// TwinCAT 3 PLC project IDPLC
// ProgramVersion: 3.1.4024.12
// libraries:
//   Tc2_Drive, * (Beckhoff Automation GmbH)
//   Tc2_EtherCAT, * (Beckhoff Automation GmbH)
//   Tc2_Math, * (Beckhoff Automation GmbH)
//   Tc2_MC2, * (Beckhoff Automation GmbH)
//   Tc2_NC, * (Beckhoff Automation GmbH)
//   Tc2_NcDrive, * (Beckhoff Automation GmbH)
//   Tc2_SerialCom, * (Beckhoff Automation GmbH)
//   Tc2_Standard, * (Beckhoff Automation GmbH)
//   Tc2_System, * (Beckhoff Automation GmbH)
//   Tc2_Utilities, * (Beckhoff Automation GmbH)
//   Tc3_Module, * (Beckhoff Automation GmbH)
// project tree:
//   DUTs/ DUT.TcDUT, DUT_SENSOR_DATAS_1.TcDUT, DUT_SENSOR_DATAS_8.TcDUT, DUT_SENSOR_DATAS_2.TcDUT, DUT_SENSOR_DATAS_3.TcDUT, DUT_SENSOR_DATAS_4.TcDUT, DUT_SENSOR_DATAS_5.TcDUT, DUT_SENSOR_DATAS_6.TcDUT, DUT_SENSOR_DATAS_7.TcDUT, Struct_M_Compensation.TcDUT, Struct_M_lakeshore.TcDUT
//   GVLs/ Global_Variables.TcGVL, Variable_Configuration.TcGVL
//   / PlcTask.TcTTO, RecipeManager.TcRMO (not stored)
//   POUs/0.UserMode/ F_GetSysTime.TcPOU, UserMode.TcPOU
//   POUs/1.CarrierMode/GapMode/ BCGapMode.TcPOU, GapMode.TcPOU
//   POUs/1.CarrierMode/SingleCarrierMode/ SingleCarrierMode.TcPOU
//   POUs/2.SingleMotorMode/DebugMode/ DebugMode.TcPOU
//   POUs/2.SingleMotorMode/TaperMode/ TaperMode.TcPOU
//   POUs/CommonFB/ExternFB/ FB_LedShow.TcPOU, FB_PlcEmergencyStop.TcPOU
//   POUs/CommonFB/MainFB/ FB_CoupleAxis.TcPOU, FB_DecoupleAxis.TcPOU, FB_Move.TcPOU, FB_Power.TcPOU, FB_SetAxisPosition.TcPOU, FB_Stop.TcPOU
//   POUs/ MAIN.TcPOU
//   POUs/MainPRG/ FB_CheckCoupleStatus.TcPOU
//   POUs/RS232/ BackgroundEL.TcPOU, FB_SerialCom.TcPOU

CONFIGURATION IDPLC
    RESOURCE PLC ON TwinCAT3
        TASK PlcTask(INTERVAL := T#10ms, PRIORITY := 20);
        PROGRAM MAIN WITH PlcTask : MAIN;
    END_RESOURCE
END_CONFIGURATION

// ---- DUTs/DUT.TcDUT
TYPE DUT :
STRUCT
	Encoder:LREAL;
	LeftTop:LREAL;
END_STRUCT
END_TYPE

// ---- DUTs/DUT_SENSOR_DATAS_1.TcDUT
TYPE DUT_SENSOR_DATAS_1 :
UNION
	data_lreal:REAL;
	data_byte:ARRAY[0..3] OF BYTE;
END_UNION
END_TYPE

// ---- DUTs/DUT_SENSOR_DATAS_8.TcDUT
TYPE DUT_SENSOR_DATAS_8 :
UNION
	data_lreal:REAL;
	data_byte:ARRAY[0..3] OF BYTE;
END_UNION
END_TYPE

// ---- DUTs/DUT_SENSOR_DATAS_2.TcDUT
TYPE DUT_SENSOR_DATAS_2 :
UNION
	data_lreal:REAL;
	data_byte:ARRAY[0..3] OF BYTE;
END_UNION
END_TYPE

// ---- DUTs/DUT_SENSOR_DATAS_3.TcDUT
TYPE DUT_SENSOR_DATAS_3 :
UNION
	data_lreal:REAL;
	data_byte:ARRAY[0..3] OF BYTE;
END_UNION
END_TYPE

// ---- DUTs/DUT_SENSOR_DATAS_4.TcDUT
TYPE DUT_SENSOR_DATAS_4 :
UNION
	data_lreal:REAL;
	data_byte:ARRAY[0..3] OF BYTE;
END_UNION
END_TYPE

// ---- DUTs/DUT_SENSOR_DATAS_5.TcDUT
TYPE DUT_SENSOR_DATAS_5 :
UNION
	data_lreal:REAL;
	data_byte:ARRAY[0..3] OF BYTE;
END_UNION
END_TYPE

// ---- DUTs/DUT_SENSOR_DATAS_6.TcDUT
TYPE DUT_SENSOR_DATAS_6 :
UNION
	data_lreal:REAL;
	data_byte:ARRAY[0..3] OF BYTE;
END_UNION
END_TYPE

// ---- DUTs/DUT_SENSOR_DATAS_7.TcDUT
TYPE DUT_SENSOR_DATAS_7 :
UNION
	data_lreal:REAL;
	data_byte:ARRAY[0..3] OF BYTE;
END_UNION
END_TYPE

// ---- DUTs/Struct_M_Compensation.TcDUT
TYPE Struct_M_Compensation :
STRUCT
	Encoder:LREAL;
	LeftTop:LREAL;
	RightTop:LREAL;
	LeftBottom:LREAL;
	RightBottom:LREAL;
	InRange:BOOL;
END_STRUCT
END_TYPE

// ---- DUTs/Struct_M_lakeshore.TcDUT
TYPE Struct_M_lakeshore :
STRUCT
	Temperature:LREAL;(*Celsius*)
	Resistance:LREAL;
END_STRUCT
END_TYPE

// ---- GVLs/Global_Variables.TcGVL
//{attribute 'Tc2GvlVarNames'}
VAR_GLOBAL
(*IDControl Ready*)
	IDControlReady:BOOL;
(*Error Massage*)
	Error:BOOL;
	ErrorID:DINT;
	ErrorDescription:STRING;
(*加载配方参数*)
	LoadRecipeParameters:BOOL;
	loadParametersDone:BOOL;
(*设置光栅bias done *)	
	PositionBiasDone:BOOL;
(*回程差*)
	HysteresisError:LREAL;
(*Drive Status*)
	DriveStatus:DINT;//1:Drive Ready;2:Axis is in operation;0:Others
(*光栅漂移误差阈值*)
	LEDriftErrorThreshold:LREAL:=0.001;
(*Lag Distance threshold*)
	PosDiff_LeftTopLin: LREAL:=0.5;
	PosDiff_RightTopLin:LREAL:=0.5;
	PosDiff_LeftBottomLin:LREAL:=0.5;
	PosDiff_RightBottomLin:LREAL:=0.5;
(*UserMode Threshold*)
	Threshold_UserTopPos: LREAL:=0.5;
	Threshold_UserBottomPos: LREAL:=0.5;
	Threshold_UserLeftPos: LREAL:=0.5;
	Threshold_UserRightPos: LREAL:=0.5;
	Threshold_UserTopVelo: LREAL:=0.5;
	Threshold_UserBottomVelo: LREAL:=0.5;
	Threshold_UserLeftVelo: LREAL:=0.5;
	Threshold_UserRightVelo: LREAL:=0.5;
	//
	Range_UserTaperPos:LREAL:=4.01;
	Range_UserTaperVelo:LREAL:=1.01;
	//Diff_TaperLeftPos:LREAL:=0.01;
	//Diff_TaperLeftVelo:LREAL:=0.2;
	//Diff_TaperRightPos:LREAL:=0.05;
	//Diff_TaperRightVelo:LREAL:=0.5;
	//Taper_BeyondRangePositive:BOOL;
	//Diff_TaperTopPos:LREAL:=0.05;
	//Diff_TaperBottomPos:LREAL:=0.05;
	//Taper_BeyondRangeNegtive:BOOL;
(*BCGap Threshold*)
	Threshold_BCTopPos: LREAL:=0.5;
	Threshold_BCBottomPos: LREAL:=0.5;
	Threshold_BCLeftPos: LREAL:=0.5;
	Threshold_BCRightPos: LREAL:=0.5;
	Threshold_BCTopVelo: LREAL:=0.5;
	Threshold_BCBottomVelo: LREAL:=0.5;
	Threshold_BCLeftVelo: LREAL:=0.5;
	Threshold_BCRightVelo: LREAL:=0.5;
(*DebugMode Threshold*)
	Threshold_TopPos_Debug: LREAL:=4;
	Threshold_BottomPos_Debug: LREAL:=4;
	Threshold_LeftPos_Debug: LREAL:=4;
	Threshold_RightPos_Debug: LREAL:=4;
(*Taper Mode Threshold*)
	Range_TaperPos:LREAL:=5.01;
	Range_TaperVelo:LREAL:=1.01;
	Threshold_TaperLeftPos:LREAL:=0.01;
	Threshold_TaperLeftVelo:LREAL:=0.2;
	Threshold_TaperRightPos:LREAL:=0.05;
	Threshold_TaperRightVelo:LREAL:=0.5;
	Taper_BeyondRangePositive:BOOL;
	Threshold_TaperTopPos:LREAL:=0.05;
	Threshold_TaperBottomPos:LREAL:=0.05;
	Taper_BeyondRangeNegtive:BOOL;
(*SingleCarrierMode threshold*)
	Threshold_TopPos_SingleCarrier: LREAL:=2;
	Threshold_BottomPos_SingleCarrier: LREAL:=2;
	Threshold_LeftPos_SingleCarrier: LREAL:=2;
	Threshold_RightPos_SingleCarrier: LREAL:=2;
	Threshold_TopVelo_SingleCarrier: LREAL:=2;
	Threshold_BottomVelo_SingleCarrier: LREAL:=2;
	Threshold_LeftVelo_SingleCarrier: LREAL:=2;
	Threshold_RightVelo_SingleCarrier: LREAL:=2;
(*Compensation Value*)
	M_Compensation:ARRAY[1..18] OF Struct_M_Compensation
:=[
(Encoder:=0,	LeftTop:=0,	RightTop:=0,		LeftBottom:=0,	RightBottom:=0,	InRange:=FALSE),
(Encoder:=5.5,	LeftTop:=5.5,	RightTop:=5.5,	LeftBottom:=5.5,	RightBottom:=5.5,	InRange:=FALSE),
(Encoder:=6.0,	LeftTop:=6.0,	RightTop:=6.0,	LeftBottom:=6.0,	RightBottom:=6.0,	InRange:=FALSE),
(Encoder:=6.5,	LeftTop:=6.5,	RightTop:=6.5,	LeftBottom:=6.5,	RightBottom:=6.5,	InRange:=FALSE),
(Encoder:=7.5,	LeftTop:=7.5,	RightTop:=7.5,	LeftBottom:=7.5,	RightBottom:=7.5,	InRange:=FALSE),
(Encoder:=8.5,	LeftTop:=8.5,	RightTop:=8.5,	LeftBottom:=8.5,	RightBottom:=8.5,	InRange:=FALSE),
(Encoder:=9.5,	LeftTop:=9.5,	RightTop:=9.5,	LeftBottom:=9.5,	RightBottom:=9.5,	InRange:=FALSE),
(Encoder:=10.5,	LeftTop:=10.5,	RightTop:=10.5,	LeftBottom:=10.5,	RightBottom:=10.5,		InRange:=FALSE),
(Encoder:=11.5,	LeftTop:=11.5,	RightTop:=11.5,	LeftBottom:=11.5,	RightBottom:=11.5,		InRange:=FALSE),
(Encoder:=30.0,	LeftTop:=30.0,	RightTop:=30.0,	LeftBottom:=30.0,	RightBottom:=30.0,		InRange:=FALSE),
(Encoder:=100.0,	LeftTop:=100.0,	RightTop:=100.0,	LeftBottom:=100.0,	RightBottom:=100.0,		InRange:=FALSE),
(Encoder:=110.0,	LeftTop:=110.0,	RightTop:=110.0,	LeftBottom:=110.0,	RightBottom:=110.0,		InRange:=FALSE),
(Encoder:=120.0,	LeftTop:=120.0,	RightTop:=120.0,	LeftBottom:=120.0,	RightBottom:=120.0,		InRange:=FALSE),
(Encoder:=130.0,	LeftTop:=130.0,	RightTop:=130.0,	LeftBottom:=130.0,	RightBottom:=130.0,		InRange:=FALSE),
(Encoder:=140.0,	LeftTop:=140.0,	RightTop:=140.0,	LeftBottom:=140.0,	RightBottom:=140.0,		InRange:=FALSE),
(Encoder:=150.0,	LeftTop:=150.0,	RightTop:=150.0,	LeftBottom:=150.0,	RightBottom:=150.0,		InRange:=FALSE),
(Encoder:=160.0,	LeftTop:=160.0,	RightTop:=160.0,	LeftBottom:=160.0,	RightBottom:=160.0,		InRange:=FALSE),
(Encoder:=3000.001,	LeftTop:=3000.001,	RightTop:=3000.001,		LeftBottom:=3000.001,	RightBottom:=3000.001,	InRange:=FALSE)];

(*simulation OR NOT*)
	simulation:BOOL;
(*USELinearEncoeder*)
	USELinearEncoder:BOOL:=TRUE;
(*restartTwinCAT*)
	m_restartTC:BOOL;
(*Plc_EmergencyStop *)
	Plc_EmergencyStop  AT %Q*:BOOL:=TRUE;
(*硬急停*)
	Hardware_EmergencyStop :BOOL:=TRUE;
(*LED*)
	Led_Run  AT %Q*:BOOL;
	Led_Error  AT %Q*:BOOL;
(*LimitSwitch*)
	LS_LeftTop_Top  :BOOL;
	LS_LeftTop_Bottom  :BOOL;
	LS_RightTop_Top  :BOOL;
	LS_RightTop_Bottom  :BOOL;
	LS_LeftBottom_Top  :BOOL;
	LS_LeftBottom_Bottom  :BOOL;
	LS_RightBottom_Top :BOOL;
	LS_RightBottom_Bottom  :BOOL;
	Unreach_LS_Top:BOOL;
	Unreach_LS_Bottom:BOOL;
(*kill switch*)
	KS_LeftTop_Far_Contact1:BOOL;
	KS_LeftTop_Far_Contact2:BOOL;
	KS_RightTop_Far_Contact1:BOOL;
	KS_RightTop_Far_Contact2:BOOL;
	KS_LeftBottom_Far_Contact1:BOOL;
	KS_LeftBottom_Far_Contact2:BOOL;
	KS_RightBottom_Far_Contact1:BOOL;
	KS_RightBottom_Far_Contact2:BOOL;
	
	KS_LeftTop_Near_Contact1:BOOL;
	KS_LeftTop_Near_Contact2:BOOL;
	KS_RightTop_Near_Contact1:BOOL;
	KS_RightTop_Near_Contact2:BOOL;
	KS_LeftBottom_Near_Contact1:BOOL;
	KS_LeftBottom_Near_Contact2:BOOL;
	KS_RightBottom_Near_Contact1:BOOL;
	KS_RightBottom_Near_Contact2:BOOL;
(*E-STOP*)
	KS_CabinetEmergency_contact1:BOOL;
	KS_CabinetEmergency_contact2:BOOL;
	KS_handEmergency1_Contact1:BOOL;
	KS_handEmergency1_Contact2:BOOL;
	KS_handEmergency2_Contact1:BOOL;
	KS_handEmergency2_Contact2:BOOL;
	KS_softEmergency2_Contact:BOOL;
(*aixs_ref*)
	LeftTopLin: axis_ref;
	RightTopLin:axis_ref;
	LeftBottomLin:axis_ref;
	RightBottomLin:axis_ref;
(*axis Position*)
	Pos_LeftTopLin: LREAL;
	Pos_RightTopLin:LREAL;
	Pos_LeftBottomLin:LREAL;
	Pos_RightBottomLin:LREAL;
(*********)
	LB_TestRecord:LREAL;
	RB_TestRecord:LREAL;
(*axis Velocity*)
	Velo_LeftTopLin: LREAL;
	Velo_RightTopLin:LREAL;
	Velo_LeftBottomLin:LREAL;
	Velo_RightBottomLin:LREAL;
(*Lag Distance*)
	PosDiff_LeftTopLin_actual: LREAL;
	PosDiff_RightTopLin_actual:LREAL;
	PosDiff_LeftBottomLin_actual:LREAL;
	PosDiff_RightBottomLin_actual:LREAL;
(********************Gap Mode*************************)
(**)
	GapPositionActual:LREAL;
	GapVelocityActual:LREAL;
	GapMoveIndicator:DINT:=0;
	(*1=OPEN;0=NOTMOVE;-1=CLOSE*)
(******************Taper Mode**************************)
(*Taper*)
	TaperPositionActual:LREAL;
	TaperVelocityActual:LREAL;
	TaperMoveIndicator:DINT:=0;
	(*1=OPEN;0=NOTMOVE;-1=CLOSE*)
(*****************singleCarrier Mode*******************************)
(**)
	TopPositionActual:LREAL;
	TopVelocityActual:LREAL;
	BottomPositionActual:LREAL;
	BottomVelocityActual:LREAL;
	TopMoveIndicator:DINT:=0;
	(*1=OPEN;0=NOTMOVE;-1=CLOSE*)
	BottomMoveIndicator:DINT:=0;
	(*1=OPEN;0=NOTMOVE;-1=CLOSE*)
(******************DebugMode & BCGapMode*****************************)
	LeftTopLinMoveIndicator:DINT:=0;
	(*1=OPEN;0=NOTMOVE;-1=CLOSE*)
	LeftBottomLinMoveIndicator:DINT:=0;
	(*1=OPEN;0=NOTMOVE;-1=CLOSE*)
	RightTopLinMoveIndicator:DINT:=0;
	(*1=OPEN;0=NOTMOVE;-1=CLOSE*)
	RightBottomLinMoveIndicator:DINT:=0;
	(*1=OPEN;0=NOTMOVE;-1=CLOSE*)
(******************Gap&SingleCarrier***********************************)
	Diff_TopPos_actual: LREAL;
	Diff_BottomPos_actual: LREAL;
	Diff_LeftPos_actual: LREAL;
	Diff_RightPos_actual: LREAL;
	Diff_TopVelo_actual:  LREAL;
	Diff_BottomVelo_actual: LREAL;
	Diff_LeftVelo_actual: LREAL;
	Diff_RightVelo_actual:  LREAL;

(******************BCGap Mode***********************************)
	Diff_BCTopPos_actual: LREAL;
	Diff_BCBottomPos_actual: LREAL;
	Diff_BCLeftPos_actual: LREAL;
	Diff_BCRightPos_actual: LREAL;
	Diff_BCTopVelo_actual:  LREAL;
	Diff_BCBottomVelo_actual: LREAL;
	Diff_BCLeftVelo_actual: LREAL;
	Diff_BCRightVelo_actual:  LREAL;
(******************UserMode*********************)
	Diff_UserTopPos_actual: LREAL;
	Diff_UserBottomPos_actual: LREAL;
	Diff_UserLeftPos_actual: LREAL;
	Diff_UserRightPos_actual: LREAL;
	Diff_UserTopVelo_actual:  LREAL;
	Diff_UserBottomVelo_actual: LREAL;
	Diff_UserLeftVelo_actual: LREAL;
	Diff_UserRightVelo_actual:  LREAL;
	TaperOrNot:BOOL;
	UserTaperPositionActual:LREAL;
	UserTaperVelocityActual:LREAL;
(***********************Power status and couple statatus***********************)
	st_Power:BOOL;
	st_Couple:DINT;
(************************FB***********************)
	FB_Power:FB_Power;
	FB_PlcEmergencyStop: FB_PlcEmergencyStop;
	FB_CheckCoupleStatus:FB_CheckCoupleStatus;
	FB_Move:FB_Move;
	FB_Stop:FB_Stop;
	FB_DecoupleAxis:FB_DecoupleAxis;
	FB_CoupleAxis: FB_CoupleAxis;
(********************²¹³¥GapÄ£Ê½£¬µ¥Öá²¹³¥Êý¾Ý************************)
	(*ÊÇ·ñ²¹³¥*)
	USE_SingleAxis_Compensation:BOOL:=TRUE;
	Mdut:ARRAY[1..2] OF DUT:=
	[(Encoder:=2.0,	LeftTop:=2.3000),
	(Encoder:=2.0,	LeftTop:=2.3000)];


	M_CompensationNumber:INT;
	M_DisplayNumber:INT;
	(*Conpensation Position Target*)
	LeftTopLinPositionNew:LREAL;
	LeftBottomLinPositionNew:LREAL;
	RightTopLinPositionNew:LREAL;
	RightBottomLinPositionNew:LREAL;
	(*考虑到回程差后，运动到临时位置*)
	LeftTopLinPositionNew_temporary :LREAL;
	LeftBottomLinPositionNew_temporary:LREAL;
	RightTopLinPositionNew_temporary:LREAL;
	RightBottomLinPositionNew_temporary:LREAL;
	(*Display Position*)
	LeftTopLinPositionDisplay:LREAL;
	LeftBottomLinPositionDisplay:LREAL;
	RightTopLinPositionDisplay:LREAL;
	RightBottomLinPositionDisplay:LREAL;
	(*Display Velocity*)
	LeftTopLinVelocityDisplay:LREAL;
	LeftBottomLinVelocityDisplay:LREAL;
	RightTopLinVelocityDisplay:LREAL;
	RightBottomLinVelocityDisplay:LREAL;
	(*temperature sensors*)
	thermocouple AT %I*:ARRAY[1..12]OF  DINT;
	shieldPt100  AT %I*:ARRAY[1..12]OF INT;
	thermocouple_Celsius:ARRAY[1..12]OF  LREAL;
	shieldPt100_Celsius  :ARRAY[1..12]OF LREAL;
	huoer_Celsius AT %I* :ARRAY[1..3]OF INT;
	(**)
	lakeshorePt100  AT %I*:ARRAY[1..12]OF INT;(*16*×èÖµ*)
	lakeshorePt100_Resistance :ARRAY[1..12]OF LREAL;(*ÉãÊÏÎÂ¶È*)
	lakeshorePt100_Celsius  :ARRAY[1..12]OF LREAL;(*ÉãÊÏÎÂ¶È*)
	temperatureCompensationValue:LREAL:=6;
	testSensors  AT %I*:ARRAY[1..4]OF INT;

(*Test No.184*)
	Struct_M_lakeshore_168:ARRAY[1..52] OF Struct_M_lakeshore:=[(Temperature:=-255.02072961,	Resistance:=19394.22709513),
														       (Temperature:=-254.05045152,	Resistance:=17654.92429047),
														       (Temperature:=-253.07744087,	Resistance:=16151.62683151),
														       (Temperature:=-252.00959324,	Resistance:=14730.57326945),
														       (Temperature:=-250.42495220,	Resistance:=12968.55015283),
														       (Temperature:=-248.82081761,	Resistance:=11509.89960915),
														       (Temperature:=-247.21174565,	Resistance:=10296.55197911),
														       (Temperature:=-245.58891366,	Resistance:=9270.75571767),
														       (Temperature:=-243.96558907,	Resistance:=8400.62569432),
														       (Temperature:=-242.14354329,	Resistance:=7573.26483503),
														       (Temperature:=-240.02689351,	Resistance:=6767.17126789),
														       (Temperature:=-237.01618411,	Resistance:=5838.58514549),
														       (Temperature:=-234.00593745,	Resistance:=5101.58555065),
														       (Temperature:=-230.99752410,	Resistance:=4505.18214539),
														       (Temperature:=-228.00173193,	Resistance:=4017.09732257),
														       (Temperature:=-224.99947745,	Resistance:=3609.02040601),
														       (Temperature:=-223.00692641,	Resistance:=3374.28026471),
														       (Temperature:=-218.01660226,	Resistance:=2884.61719537),
														       (Temperature:=-213.02574325,	Resistance:=2501.58514940),
														       (Temperature:=-208.03560884,	Resistance:=2195.64012040),
														       (Temperature:=-203.04420176,	Resistance:=1946.81103230),
														       (Temperature:=-198.05275449,	Resistance:=1741.06206884),
														       (Temperature:=-193.06103279,	Resistance:=1568.92560629),
														       (Temperature:=-188.06248282,	Resistance:=1422.92395120),
														       (Temperature:=-183.06714354,	Resistance:=1298.17958491),
														       (Temperature:=-178.06870827,	Resistance:=1190.47468069),
														       (Temperature:=-173.07068956,	Resistance:=1096.60468916),
														       (Temperature:=-163.08053594,	Resistance:=942.07281950),
														       (Temperature:=-153.08718985,	Resistance:=820.42837839),
														       (Temperature:=-143.08487641,	Resistance:=722.56760466),
														       (Temperature:=-133.08398781,	Resistance:=642.67848926),
														       (Temperature:=-123.08745222,	Resistance:=576.45895597),
														       (Temperature:=-113.09120089,	Resistance:=520.90762376),
														       (Temperature:=-103.09942915,	Resistance:=473.74837218),
														       (Temperature:=-93.10598968,		Resistance:=433.38294834),
														       (Temperature:=-83.10392915,		Resistance:=398.41968464),
														       (Temperature:=-73.10228709,		Resistance:=368.09301028),
														       (Temperature:=-63.10299621,		Resistance:=341.43424414),
														       (Temperature:=-53.11519681,		Resistance:=318.02847824),
														       (Temperature:=-43.10742807	,	Resistance:=297.22485607),
														       (Temperature:=-33.10726812,		Resistance:=278.69871028),
														       (Temperature:=-23.11858134,		Resistance:=262.15834948),
														       (Temperature:=-13.10195090,		Resistance:=247.23616978),
														       (Temperature:=-3.11184252,		Resistance:=233.79708047),
														       (Temperature:=6.89903472,		Resistance:=221.61300733),
														       (Temperature:=16.89346621,		Resistance:=210.54967929),
														       (Temperature:=26.90358952,		Resistance:=200.45587628),
														       (Temperature:=36.88287604,		Resistance:=191.25204791),
														       (Temperature:=41.88872196,		Resistance:=186.92616816),
														       (Temperature:=46.88480694,		Resistance:=182.78432099),
														       (Temperature:=52.87776550,		Resistance:=178.06184409),
														       (Temperature:=56.87370113,		Resistance:=175.01081354)];

(*
Struct_M_lakeshore_168:ARRAY[1..52] OF Struct_M_lakeshore:=(Temperature:=-255.02148584,	Resistance:=17467.51361429),
														       (Temperature:=-254.05229765,	Resistance:=15920.82205731),
														       (Temperature:=-253.07582822,	Resistance:=14578.50586503),
														       (Temperature:=-252.01029408,	Resistance:=13314.83293750),
														       (Temperature:=-250.42593953,	Resistance:=11741.46150061),
														       (Temperature:=-248.82114671,	Resistance:=10435.92048251),
														       (Temperature:=-247.21093179,	Resistance:=9348.73725539),
														       (Temperature:=-245.58869114,	Resistance:=8428.36508630),
														       (Temperature:=-243.96317077,	Resistance:=7645.95382882),
														       (Temperature:=-242.14282659,	Resistance:=6901.52980185),
														       (Temperature:=-240.02565306,	Resistance:=6174.70288700),
														       (Temperature:=-237.01772619,	Resistance:=5337.15935418),
														       (Temperature:=-234.00641032,	Resistance:=4669.94432605),
														       (Temperature:=-230.99638631,	Resistance:=4129.44762482),
														       (Temperature:=-228.00091359,	Resistance:=3686.25091590),
														       (Temperature:=-225.00020456,	Resistance:=3315.69773718),
														       (Temperature:=-223.00791577,	Resistance:=3102.03825436),
														       (Temperature:=-218.01784455,	Resistance:=2655.95765650),
														       (Temperature:=-213.02820409,	Resistance:=2306.30469335),
														       (Temperature:=-208.03707086,	Resistance:=2026.68631979),
														       (Temperature:=-203.04413996,	Resistance:=1798.75031171),
														       (Temperature:=-198.05551086,	Resistance:=1610.35975891),
														       (Temperature:=-193.06273927,	Resistance:=1452.39526661),
														       (Temperature:=-188.05883288,	Resistance:=1318.25592597),
														       (Temperature:=-183.06258538,	Resistance:=1203.56234118),
														       (Temperature:=-178.06718279,	Resistance:=1104.51148216),
														       (Temperature:=-173.07249199,	Resistance:=1018.20332165),
														       (Temperature:=-163.08375191,	Resistance:=875.68114167),
														       (Temperature:=-153.08708895,	Resistance:=763.40014611),
														       (Temperature:=-143.08456026,	Resistance:=673.01413079),
														       (Temperature:=-133.08511977,	Resistance:=599.14558137),
														       (Temperature:=-123.08749266,	Resistance:=537.87435730),
														       (Temperature:=-113.09351200,	Resistance:=486.39730699),
														       (Temperature:=-103.10083499,	Resistance:=442.70701049),
														       (Temperature:=-93.10681179,		Resistance:=405.24490154),
														       (Temperature:=-83.10668364,		Resistance:=372.85251196),
														       (Temperature:=-73.10424427,		Resistance:=344.62377216),
														       (Temperature:=-63.10525050,		Resistance:=319.91272482),
														       (Temperature:=-53.11631884,		Resistance:=298.14326645),
														       (Temperature:=-43.10919062	,	Resistance:=278.79776489),
														       (Temperature:=-33.10718139,		Resistance:=261.57224548),
														       (Temperature:=-23.12143823,		Resistance:=246.17864217),
														       (Temperature:=-13.10564070,		Resistance:=232.27707124),
														       (Temperature:=-3.11271856,		Resistance:=219.77787693),
														       (Temperature:=6.89876028,		Resistance:=208.41568062),
														       (Temperature:=16.88935188,		Resistance:=198.10158580),
														       (Temperature:=26.89992337,		Resistance:=188.70405160),
														       (Temperature:=36.88110394,		Resistance:=180.10572832),
														       (Temperature:=41.88616228,		Resistance:=176.08361784),
														       (Temperature:=46.88372409,		Resistance:=172.21346348),
														       (Temperature:=52.87452959,		Resistance:=167.80352164),
														       (Temperature:=56.87233822,		Resistance:=164.96790544);
*)

(******RS232************)
	RxBufferEL			: ComBuffer;	(* Receive data buffer; used with all receive function blocks *)
	TxBufferEL			: ComBuffer;	(* Transmit data buffer; used with all receive function blocks *)

END_VAR

// ---- GVLs/Variable_Configuration.TcGVL
{attribute 'Tc2GvlVarNames'}
VAR_CONFIG
END_VAR

// ---- POUs/MAIN.TcPOU
PROGRAM MAIN
VAR
	pbGapMode: BOOL:=FALSE;
	pbTaperMode: BOOL:=FALSE;
	pbSingleCarrierMode: BOOL:=FALSE;
	pbDebugMode:BOOL:=FALSE;
	pbBCGapMode:BOOL:=FALSE;
	fb_led_Show: FB_LedShow;
	btn_reset: BOOL;
	CPMU_PLC_Reset: PLC_Reset;
	d_state: DINT;
	CPMU_PLC_Start: PLC_Start;
	powerStatus:BOOL;

(*TwinSAFE*)
	Safe_run AT%Q*:BOOL;
	Err_Ack AT %Q*:BOOL;
	Estop_RunAndRestart AT %Q*:BOOL;
	AX5805_Error_Ack AT %Q*:BOOL;
	Led_Run  AT %Q*:BOOL;
	Led_Error  AT %Q*:BOOL;

	FB_ERROR AT%I*:BOOL;
	COM_ERROR AT%I*:BOOL;
	//OUT_ERROR AT%I*:BOOL;
	Estop_Out AT%I*:BOOL;

	SafeStatus:INT;
	SafePLCRunOK: BOOL;
	fb_ton: TON;
	fb_ton2: TON;
	fb_ton3: TON;
	fb_ton1: TON;
	fb_ton0: TON;
(*IO*)
	el1808_D1  AT%I* :ARRAY[1..8] OF BOOL;
	el1008 AT%I*:BOOL;
	EStopTrig:BOOL;
(*setAxisPosition*)
	SetAxisPosState: INT;
	FB_Set_AxisPosition:FB_SetAxisPosition;
	fb_ton4: TON;
	fb_ton5: TON;
	fb_ton6: TON;
	SerAxisPositionDone: BOOL;

	i: INT;
	j: INT;

(****RS232***)
	fbEL6001	: FB_SerialCom;
	moveDoneLeftTop: BOOL;
	moveDoneRightTop: BOOL;
	moveDoneLeftBottom: BOOL;
	moveDoneRightBottom: BOOL;
	moveDoneAllAxis: BOOL;
	moveStatusLeftTop: BOOL;
	moveStatusRightTop: BOOL;
	moveStatusLeftBottom: BOOL;
	moveStatusRightBottom: BOOL;
	moveStatusAllAxis: BOOL;

(*Torque*)
	Torque_LT AT%I*:INT;
	Torque_RT AT%I*:INT;
	Torque_LB AT%I*:INT;
	Torque_RB AT%I*:INT;
(**)
	btn_setAxisPosition: BOOL;
	ValueSet_LeftTop:LREAL;
	ValueSet_RightTop:LREAL;
	ValueSet_LeftBottom:LREAL;
	ValueSet_RightBottom:LREAL;
(**)
	RestartTC: TC_Restart;
	
(*recipe*)
	RecipeINT:INT;
	RecipeBOOL:BOOL;
	RecipeManCommands: RecipeManCommands;
	SaveParameter : BOOL;  //保存文件
	LoadParameter : BOOL;  //读取文件
	Save_R_TRIG   : R_TRIG;
	Read_R_TRIG   : R_TRIG;
	loadparameterStatus: INT;
	RecipeBOOL2:BOOL;
	ReturnDwordLoad: DWORD;
	InsertionDeviceName:STRING;
(*UserMode*)
	pbUserMode: BOOL:=TRUE;
	EL1904 AT%I* :ARRAY[1..24] OF BOOL;
	setAxisPositionEnable: BOOL;
	state_loadParameters: INT;
	state_setLEPosBias: INT;
	//
	PositionBiasSet:BOOL;
	MC_SetLEPosBias_LeftTop:MC_WriteParameter;
	MC_SetLEPosBias_RightTop:MC_WriteParameter;
	MC_SetLEPosBias_LeftBottom:MC_WriteParameter;
	MC_SetLEPosBias_RightBottom:MC_WriteParameter;
	PositionBias_LeftTop: LREAL:=10.1;
	PositionBias_RightTop: LREAL:=10.2;
	PositionBias_LeftBottom: LREAL:=10.3;
	PositionBias_RightBottom: LREAL:=10.4;

	LoadLEPB_R_TRIG: R_TRIG;
	PositionBiasTON: TON;
	
	//
	OPC_TEST_Bi:BOOL:=TRUE; (*~ (OPC:1:available for OPC Clients) *)
	OPC_TEST_Bi2:BOOL;(*~ (OPC:1:available for OPC Clients) *)
	//
	HasTemperatureSensorOrNot:BOOL;//Only IVU or CPMU
	(*Sensor Reading*)
	Sensor_Reading_1 AT %I*:ARRAY[0..3] OF BYTE;
	Sensor_Reading_2 AT %I*:ARRAY[0..3] OF BYTE;
	Sensor_Reading_3 AT %I*:ARRAY[0..3] OF BYTE;
	Sensor_Reading_4 AT %I*:ARRAY[0..3] OF BYTE;
	Sensor_Reading_5 AT %I*:ARRAY[0..3] OF BYTE;
	Sensor_Reading_6 AT %I*:ARRAY[0..3] OF BYTE;
	Sensor_Reading_7 AT %I*:ARRAY[0..3] OF BYTE;
	Sensor_Reading_8 AT %I*:ARRAY[0..3] OF BYTE;
	Sensor_Reading_DpState AT %I*:USINT;
	Sensor_Reading_ExtDiagFlag AT %I*:BOOL;
	TemperatureSensors_1:LREAL;
	TemperatureSensors_2:LREAL;
	TemperatureSensors_3:LREAL;
	TemperatureSensors_4:LREAL;
	TemperatureSensors_5:LREAL;
	TemperatureSensors_6:LREAL;
	TemperatureSensors_7:LREAL;
	TemperatureSensors_8:LREAL;
	dut_sensor_datas_1:DUT_SENSOR_DATAS_1;
	dut_sensor_datas_2:DUT_SENSOR_DATAS_2;
	dut_sensor_datas_3:DUT_SENSOR_DATAS_3;
	dut_sensor_datas_4:DUT_SENSOR_DATAS_4;
	dut_sensor_datas_5:DUT_SENSOR_DATAS_5;
	dut_sensor_datas_6:DUT_SENSOR_DATAS_6;
	dut_sensor_datas_7:DUT_SENSOR_DATAS_7;
	dut_sensor_datas_8:DUT_SENSOR_DATAS_8;
	//
	temperature_gradient_2_To_1:LREAL;
	temperature_gradient_3_To_2:LREAL;
	temperature_gradient_5_To_4:LREAL;
	temperature_gradient_6_To_5:LREAL;
	temperature_gradient_max:LREAL;
	//
	temperature_average:LREAL;
	A_SetLinearEncoderPositionBias_Enable: BOOL;
	
		//
	temperatureStatus:INT;//0：有传感器度数错误；1:常温；2:低温；3:常温和低温中间态
	CryogenicTemperatureThreshold:LREAL:=80;//80K以下归划分为低温
	RoomTemperatureThreshold:LREAL:=293;//293K以上划分为常温
	//CPMU cryogenix ON/FF
	CryogenicCompensationOn:BOOL;
	CryogenicCompensationConditionsReady:BOOL;
	CryogenicCompensation_LeftTop:LREAL;
	CryogenicCompensation_RightTop:LREAL;
	CryogenicCompensation_LeftBottom:LREAL;
	CryogenicCompensation_RightBottom:LREAL;
	CryogenicCompensationDone: BOOL;
	
	(**)
	bDriveDiagMessageAndNumber  : BOOL;
	m_GetDriveStatusState:INT;
	GetDriveStatusStateDone:BOOL;
	GetDriveStatusStateError:BOOL;
	GetDriveStatusTON: TON;
	//	
	fb_SoEReadDiagMessage_LeftTop: FB_SoEReadDiagMessage;
	fb_SoEReadDiagMessage_RightTop: FB_SoEReadDiagMessage;
	fb_SoEReadDiagMessage_LeftBottom: FB_SoEReadDiagMessage;
	fb_SoEReadDiagMessage_RightBottom: FB_SoEReadDiagMessage;
	DriveDiagMessage_LeftTop:STRING;
	DriveDiagMessage_RightTop:STRING;
	DriveDiagMessage_LeftBottom:STRING;
	DriveDiagMessage_RightBottom:STRING;
	//
	FB_SoEReadDiagNumber_LeftTop: FB_SoEReadDiagNumber;
	FB_SoEReadDiagNumber_RightTop: FB_SoEReadDiagNumber;
	FB_SoEReadDiagNumber_LeftBottom: FB_SoEReadDiagNumber;
	FB_SoEReadDiagNumber_RightBottom: FB_SoEReadDiagNumber;
	DriveDiagNumber_LeftTop:UDINT;
	DriveDiagNumber_RightTop:UDINT;
	DriveDiagNumber_LeftBottom:UDINT;
	DriveDiagNumber_RightBottom:UDINT;
	bReloadDriveDiagMessageAndNumber: BOOL;
	
	(*load IOC*)
	bExe_load_Prog: BOOL;
	NT_StartProcess_Load: NT_StartProcess;
	Exe_load_step: UINT;
	R_TRIG_ExeLoad: R_TRIG;
	Exe_Load_Done:BOOL;
	(*kill IOC*)
	bExe_Kill_Prog: BOOL;
	NT_StartProcess_Kill: NT_StartProcess;
	Exe_kill_step: UINT;
	R_TRIG_Exekill: R_TRIG;
	Exe_Kill_Done:BOOL;
	LoadOpcIocTON:TON;
END_VAR

(*加载Ricipe参数*)
A_InitRecipeParameters();
(*Restart TwinCAT*)
IF Global_Variables.m_restartTC THEN
(*首先关闭opcIocShell.exe*)	
	bExe_Kill_Prog:=TRUE;
	A_KillOpcIocShellExe();
(*重启TC*)
	IF Exe_Kill_Done THEN
		A_RestartTC();
	END_IF
END_IF
(*******InitAxisParameters*******)
A_InitAxisParameters();
(*******CheckLimitSwitch*******)
A_CheckLimitSwitch();
(*Check Kill Switch*)
A_CheckKillSwitch();
(*******PosDiff¼à¿Ø*******)
A_PosDiffDetectiion();
(*******³õÊ¼»¯SafePlc*******)
IF NOT simulation THEN
A_SafePlcStartInit();
END_IF
(************SetAxisPosition*********************)
IF  NOT USELinearEncoder AND setAxisPositionEnable AND btn_setAxisPosition THEN
	//IF NOT SerAxisPositionDone THEN
		FB_Set_AxisPosition.ValueSet_LeftTop:=ValueSet_LeftTop;
		FB_Set_AxisPosition.ValueSet_RightTop:=ValueSet_RightTop;
		FB_Set_AxisPosition.ValueSet_LeftBottom:=ValueSet_LeftBottom;
		FB_Set_AxisPosition.ValueSet_RightBottom:=ValueSet_RightBottom;
		A_SetAxisPosition();
	//END_IF
END_IF
(*******³Mode Select******)
IF SafePLCRunOK OR Simulation THEN
	IF pbSingleCarrierMode AND NOT pbTaperMode AND NOT pbGapMode AND NOT pbDebugMode AND NOT pbBCGapMode AND NOT pbUserMode THEN
		SingleCarrierMode();
	ELSIF pbTaperMode  AND NOT pbSingleCarrierMode AND NOT pbGapMode  AND NOT pbDebugMode AND NOT pbBCGapMode AND NOT pbUserMode THEN
		TaperMode();
	ELSIF pbGapMode AND  NOT pbSingleCarrierMode AND NOT pbTaperMode  AND NOT pbDebugMode AND NOT pbBCGapMode AND NOT pbUserMode THEN
		GapMode();
	ELSIF pbDebugMode AND NOT pbGapMode AND NOT pbSingleCarrierMode AND NOT pbTaperMode AND NOT pbBCGapMode  AND NOT pbUserMode THEN
		DebugMode();
	ELSIF pbBCGapMode AND NOT pbGapMode AND NOT pbSingleCarrierMode AND NOT pbTaperMode AND NOT pbDebugMode AND NOT pbUserMode THEN
		BCGapMode();
	ELSIF pbUserMode AND NOT pbGapMode AND NOT pbSingleCarrierMode AND NOT pbTaperMode AND NOT pbDebugMode AND NOT pbBCGapMode THEN
		UserMode();
	END_IF
END_IF
(*******Led Show******)
fb_led_Show();
(*******Check Power status******)
FB_Power(Check:=TRUE);
st_Power:=FB_Power.PowerState;
(******Check Couple Status*****)
FB_CheckCoupleStatus(Check:=TRUE);
st_Couple:=FB_CheckCoupleStatus.CoupleState;
(*********RS232*********************)
BackgroundEL();
(*fbEL6001(TxBuffer:=TxBufferEL, RxBuffer:=RxBufferEL);*)

(*获取温度传感器数据*)
A_GetTemperatureSensorsData();
(*低温补偿监控*)
A_CryogenicCompensationMonitoring();

(*设置position bias*)
IF loadParametersDone AND (DriveStatus=1 OR simulation) THEN 
	A_SetLinearEncoderPositionBias();
END_IF
(*检查硬急停状态，包括安全限位、柜门急停、手持急停*)
A_CheckHardwareEmergencyStopStatus();
(*获取驱动器状态信息*)
IF NOT simulation THEN
	A_GetDriverStatus();
END_IF
(*IDControlReady*)
IF ((DriveStatus<>0 AND SafePLCRunOK) OR simulation) AND NOT Error THEN
//IF (SafePLCRunOK OR simulation) AND NOT Error THEN
	IDControlReady:=TRUE;
ELSE
	IDControlReady:=FALSE;
END_IF

(*IOC Start*)
IF SafePLCRunOK OR simulation THEN
	bExe_load_Prog:=TRUE;
	A_LoadOpcIocShellExe();
END_IF

ACTION A_CheckHardwareEmergencyStopStatus:
IF 	NOT KS_LeftTop_Far_Contact1 OR
	NOT KS_LeftTop_Far_Contact2 OR
	NOT KS_RightTop_Far_Contact1 OR
	NOT KS_RightTop_Far_Contact2 OR
	NOT KS_LeftBottom_Far_Contact1 OR
	NOT KS_LeftBottom_Far_Contact2 OR
	NOT KS_RightBottom_Far_Contact1 OR
	NOT KS_RightBottom_Far_Contact2 OR
	
	NOT KS_LeftTop_Near_Contact1 OR
	NOT KS_LeftTop_Near_Contact2 OR
	NOT KS_RightTop_Near_Contact1 OR
	NOT KS_RightTop_Near_Contact2 OR
	NOT KS_LeftBottom_Near_Contact1 OR
	NOT KS_LeftBottom_Near_Contact2 OR
	NOT KS_RightBottom_Near_Contact1 OR
	NOT KS_RightBottom_Near_Contact2 OR
(*E-STOP*)
	NOT KS_CabinetEmergency_contact1 OR
	NOT KS_CabinetEmergency_contact2 OR
	NOT KS_handEmergency1_Contact1 OR
	NOT KS_handEmergency1_Contact2 OR
	NOT KS_handEmergency2_Contact1 OR
	NOT KS_handEmergency2_Contact2 OR
	NOT KS_softEmergency2_Contact THEN
	Hardware_EmergencyStop:=FALSE;
ELSE
	Hardware_EmergencyStop:=TRUE;
END_IF
END_ACTION

ACTION A_CheckKillSwitch:
IF simulation THEN
	KS_LeftTop_Far_Contact1:=TRUE;
	KS_LeftTop_Far_Contact2:=TRUE;
	KS_LeftTop_Near_Contact1:=TRUE;
	KS_LeftTop_Near_Contact2:=TRUE;
	KS_RightTop_Far_Contact1:=TRUE;
	KS_RightTop_Far_Contact2:=TRUE;
	KS_RightTop_Near_Contact1:=TRUE;
	KS_RightTop_Near_Contact2:=TRUE;
	KS_LeftBottom_Far_Contact1:=TRUE;
	KS_LeftBottom_Far_Contact2:=TRUE;
	KS_LeftBottom_Near_Contact1:=TRUE;
	KS_LeftBottom_Near_Contact2:=TRUE;	
	KS_RightBottom_Far_Contact1:=TRUE;
	KS_RightBottom_Far_Contact2:=TRUE;
	KS_RightBottom_Near_Contact1:=TRUE;
	KS_RightBottom_Near_Contact2:=TRUE;		
	(*E-STOP*)
	KS_CabinetEmergency_contact1:=TRUE;
	KS_CabinetEmergency_contact2:=TRUE;	
	KS_handEmergency1_Contact1:=TRUE;
	KS_handEmergency1_Contact2:=TRUE;
	KS_handEmergency2_Contact1:=TRUE;
	KS_handEmergency2_Contact2:=TRUE;
	
	KS_softEmergency2_Contact:=TRUE;

ELSE
	KS_LeftTop_Far_Contact1:=EL1904[1];//c1
	KS_LeftTop_Far_Contact2:=EL1904[2];//c2
	KS_LeftTop_Near_Contact1:=EL1904[3];//c3
	KS_LeftTop_Near_Contact2:=EL1904[4];//c4
	
	KS_RightTop_Far_Contact1:=EL1904[5];
	KS_RightTop_Far_Contact2:=EL1904[6];
	KS_RightTop_Near_Contact1:=EL1904[7];
	KS_RightTop_Near_Contact2:=EL1904[8];
	
	KS_LeftBottom_Far_Contact1:=EL1904[9];
	KS_LeftBottom_Far_Contact2:=EL1904[10];
	KS_LeftBottom_Near_Contact1:=EL1904[11];
	KS_LeftBottom_Near_Contact2:=EL1904[12];
	
	KS_RightBottom_Far_Contact1:=EL1904[13];
	KS_RightBottom_Far_Contact2:=EL1904[14];
	KS_RightBottom_Near_Contact1:=EL1904[15];
	KS_RightBottom_Near_Contact2:=EL1904[16];	
	
	
	(*E-STOP*)
	KS_CabinetEmergency_contact1:=EL1904[17];
	KS_CabinetEmergency_contact2:=EL1904[18];
	
	KS_handEmergency1_Contact1:=EL1904[19];
	KS_handEmergency1_Contact2:=EL1904[20];
	KS_handEmergency2_Contact1:=EL1904[21];
	KS_handEmergency2_Contact2:=EL1904[22];
	
	KS_softEmergency2_Contact:=EL1904[23];
	END_IF
END_ACTION

ACTION A_CheckLimitSwitch:
(*******1.´ÓIO»ñÈ¡ÏÞÎ»×´Ì¬******)
(**)
IF simulation THEN
	(**)
	LS_LeftTop_Top:=TRUE;
	LS_LeftTop_Bottom:=TRUE;
	LS_RightTop_Top:=TRUE;
	LS_RightTop_Bottom:=TRUE;
	LS_LeftBottom_Top:=TRUE;
	LS_LeftBottom_Bottom:=TRUE;
	LS_RightBottom_Top:=TRUE;
	LS_RightBottom_Bottom:=TRUE;
ELSE
	LS_LeftTop_Top :=el1808_D1[1];
	LS_LeftTop_Bottom:=el1808_D1[3];
	LS_RightTop_Top:=el1808_D1[2];
	LS_RightTop_Bottom:=el1808_D1[4];
	LS_LeftBottom_Top:=el1808_D1[7];
	LS_LeftBottom_Bottom:=el1808_D1[5];
	LS_RightBottom_Top:=el1808_D1[8];
	LS_RightBottom_Bottom:=el1808_D1[6];
END_IF
(*
	LS_LeftTop_Top:=TRUE;
	LS_LeftTop_Bottom:=TRUE;
	LS_RightTop_Top:=TRUE;
	LS_RightTop_Bottom:=TRUE;
	LS_LeftBottom_Top:=TRUE;
	LS_LeftBottom_Bottom:=TRUE;
	LS_RightBottom_Top:=TRUE;
	LS_RightBottom_Bottom:=TRUE;
*)
(******2.TopÏÞÎ»»òÕßBottomÏÞÎ»ÓÐÒ»¸ö´¥·¢£¬È«¾Ö±äÁ¿¡£¸øMC_POWERÓÃÓÚ·½Ïò¿ØÖÆ£¬ÓÐÒ»¸öÏÞÎ»Îª´¥·¢ÎªFALSE£¬ÔòUnreach_LSÎªFALSE******)
Unreach_LS_Top:=LS_LeftTop_Top AND LS_RightTop_Top AND LS_LeftBottom_Top AND LS_RightBottom_Top;
Unreach_LS_Bottom:=LS_LeftTop_Bottom AND LS_RightTop_Bottom AND LS_LeftBottom_Bottom AND LS_RightBottom_Bottom;
(**************************ÏòTopÔË¶¯Ê±£¬´¥ÅöBottomÏÞÎ»¿ª¹Ø£¬»òÕßÏà·´£¬ESTOP**************************************)
(*
IF LeftTopLin.Status.Moving AND Velo_LeftTopLin>0 THEN
	IF NOT Unreach_LS_Bottom THEN
		Error:=TRUE;
		ErrorID:=61;
		FB_PlcEmergencyStop();
	END_IF
ELSIF LeftTopLin.Status.Moving AND Velo_LeftTopLin<0 THEN
	IF NOT Unreach_LS_Top THEN
		Error:=TRUE;
		ErrorID:=62;
		FB_PlcEmergencyStop();
	END_IF
ELSIF RightTopLin.Status.Moving AND Velo_RightTopLin>0 THEN
	IF NOT Unreach_LS_Bottom THEN
		Error:=TRUE;
		ErrorID:=63;
		FB_PlcEmergencyStop();
	END_IF
ELSIF RightTopLin.Status.Moving AND Velo_RightTopLin<0 THEN
	IF NOT  Unreach_LS_Top THEN
		Error:=TRUE;
		ErrorID:=64;
		FB_PlcEmergencyStop();
	END_IF
ELSIF LeftBottomLin.Status.Moving AND Velo_LeftBottomLin>0 THEN
	IF NOT Unreach_LS_Bottom THEN
		Error:=TRUE;
		ErrorID:=65;
		FB_PlcEmergencyStop();
	END_IF
ELSIF LeftBottomLin.Status.Moving AND Velo_LeftBottomLin<0 THEN
	IF NOT Unreach_LS_Top THEN
		Error:=TRUE;
		ErrorID:=66;
		FB_PlcEmergencyStop();
	END_IF
ELSIF RightBottomLin.Status.Moving AND Velo_RightBottomLin>0 THEN
	IF NOT Unreach_LS_Bottom THEN
		Error:=TRUE;
		ErrorID:=67;
		FB_PlcEmergencyStop();
	END_IF
ELSIF RightBottomLin.Status.Moving AND Velo_RightBottomLin<0 THEN
	IF NOT Unreach_LS_Top THEN
		Error:=TRUE;
		ErrorID:=68;
		FB_PlcEmergencyStop();
	END_IF
END_IF
*)
(*
(******3.ÓÐÒ»¸öÏÞÎ»´¥·¢£¬ delayÊ±¼äºó£¬¼à²âÖáÊÇ·ñÔÚÍ£Ö¹×´Ì¬£¬ÈôÃ»ÓÐ£¬Emergency AND PowerOff******)
IF NOT Unreach_LS_Top OR NOT Unreach_LS_Bottom THEN
	fb_ton.IN:=TRUE;
END_IF
IF fb_ton.Q THEN
	IF LeftTopLin.Status.Moving OR RightTopLin.Status.Moving OR LeftBottomLin.Status.Moving OR RightBottomLin.Status.Moving THEN
		FB_PlcEmergencyStop();
		fb_ton.IN:=FALSE;
		Error:=TRUE;
		EStopTrig:=TRUE;
		ErrorID:=1;
		(*FB_Power_Off(Execute:=TRUE);*)
	END_IF
END_IF

(*******4.µ¥ÖáÉÏÏÂÏÞÎ»¾ùÎªFALSEÊ±£¬ÏÞÎ»´íÎó£¬Emergency*******)
IF (NOT LS_LeftTop_Top AND NOT LS_LeftTop_Bottom) OR  (NOT  LS_RightTop_Top AND NOT LS_RightTop_Bottom)
		OR (NOT LS_LeftBottom_Top AND NOT LS_LeftBottom_Bottom) OR (NOT LS_RightBottom_Top AND NOT LS_RightBottom_Bottom) THEN
	(*FB_Plc_EmergencyStop();*)
	Error:=TRUE;
	EStopTrig:=TRUE;
	ErrorID:=2;
END_IF
*)
END_ACTION

ACTION A_CryogenicCompensationMonitoring:
//没有传感器OR不是CPMU不低温补偿OR低温不到位，均不补偿
IF NOT HasTemperatureSensorOrNot OR NOT CryogenicCompensationOn THEN //OR temperatureStatus<>2 THEN
	//不补偿
	CryogenicCompensation_LeftTop:=0;
	CryogenicCompensation_RightTop:=0;
	CryogenicCompensation_LeftBottom:=0;
	CryogenicCompensation_RightBottom:=0;
ELSE
	CryogenicCompensationConditionsReady:=TRUE;//条件具备，可以低温补偿
	//检查补偿值，单轴补偿范围均在0-1内
	IF CryogenicCompensation_LeftTop>1 OR CryogenicCompensation_LeftTop<=0 THEN
			Error:=TRUE;
			ErrorID:=1201;
			ErrorDescription:='CryogenicCompensation_LeftTop>1 OR CryogenicCompensation_LeftTop<=0';
			FB_PlcEmergencyStop();
	END_IF
	IF CryogenicCompensation_RightTop>1 OR CryogenicCompensation_RightTop<=0 THEN
			Error:=TRUE;
			ErrorID:=1202;
			ErrorDescription:='CryogenicCompensation_RightTop>1 OR CryogenicCompensation_RightTop<=0';
			FB_PlcEmergencyStop();
	END_IF
	IF CryogenicCompensation_LeftBottom>1 OR CryogenicCompensation_LeftBottom<=0 THEN
			Error:=TRUE;
			ErrorID:=1203;
			ErrorDescription:='CryogenicCompensation_LeftBottom>1 OR CryogenicCompensation_LeftBottom<=0';
			FB_PlcEmergencyStop();
	END_IF
	IF CryogenicCompensation_RightBottom>1 OR CryogenicCompensation_RightBottom<=0 THEN
			Error:=TRUE;
			ErrorID:=1204;
			ErrorDescription:='CryogenicCompensation_RightBottom>1 OR CryogenicCompensation_RightBottom<=0';
			FB_PlcEmergencyStop();
	END_IF
END_IF
//若在低温补偿模式，但是温度没到低温区间，则Emergency，不允许启动
(*
IF CryogenicCompensationOn AND temperatureStatus<>2 THEN
			Error:=TRUE;
			ErrorID:=1205;
			ErrorDescription:='CryogenicCompensationOn AND temperatureStatus<>2';
			FB_PlcEmergencyStop();
END_IF
*)
END_ACTION

ACTION A_GetDriverStatus:
IF bReloadDriveDiagMessageAndNumber THEN
	m_GetDriveStatusState:=0;
	bReloadDriveDiagMessageAndNumber:=FALSE;
END_IF
GetDriveStatusTON(PT:=T#1S);
A_GetDriverStatusMC();
CASE m_GetDriveStatusState OF
	0:
		GetDriveStatusTON.IN:=TRUE;
		m_GetDriveStatusState:=1;
	1:
		IF GetDriveStatusTON.Q THEN
			bDriveDiagMessageAndNumber:=TRUE;
			m_GetDriveStatusState:=2;
		END_IF
	2:
		GetDriveStatusTON.IN:=FALSE;
		DriveDiagMessage_LeftTop:=fb_SoEReadDiagMessage_LeftTop.sDiagMessage.strData;
		DriveDiagMessage_RightTop:=fb_SoEReadDiagMessage_RightTop.sDiagMessage.strData;
		DriveDiagMessage_LeftBottom:=fb_SoEReadDiagMessage_LeftBottom.sDiagMessage.strData;
		DriveDiagMessage_RightBottom:=fb_SoEReadDiagMessage_RightBottom.sDiagMessage.strData;
		//
		DriveDiagNumber_LeftTop:=FB_SoEReadDiagNumber_LeftTop.iDiagNumber;
		DriveDiagNumber_RightTop:=FB_SoEReadDiagNumber_RightTop.iDiagNumber;
		DriveDiagNumber_LeftBottom:=FB_SoEReadDiagNumber_LeftBottom.iDiagNumber;
		DriveDiagNumber_RightBottom:=FB_SoEReadDiagNumber_RightBottom.iDiagNumber;
		//
		IF 	NOT fb_SoEReadDiagMessage_LeftTop.bBusy
			AND NOT fb_SoEReadDiagMessage_RightTop.bBusy
			AND NOT fb_SoEReadDiagMessage_LeftBottom.bBusy
			AND NOT fb_SoEReadDiagMessage_RightBottom.bBusy 
			AND NOT FB_SoEReadDiagNumber_LeftTop.bBusy
			AND NOT  FB_SoEReadDiagNumber_RightTop.bBusy
			AND NOT FB_SoEReadDiagNumber_LeftBottom.bBusy
			AND NOT FB_SoEReadDiagNumber_RightBottom.bBusy THEN
			m_GetDriveStatusState:=88;
		END_IF
		IF 	fb_SoEReadDiagMessage_LeftTop.bError
			OR fb_SoEReadDiagMessage_RightTop.bError
			OR fb_SoEReadDiagMessage_LeftBottom.bError
			OR fb_SoEReadDiagMessage_RightBottom.bError
			OR FB_SoEReadDiagNumber_LeftTop.bError
			OR FB_SoEReadDiagNumber_RightTop.bError
			OR FB_SoEReadDiagNumber_LeftBottom.bError
			OR FB_SoEReadDiagNumber_RightBottom.bError THEN
			m_GetDriveStatusState:=-100;
		END_IF
		(*Drive Status*)
		//D012, Axis state machine: Control and power section ready
		IF DriveDiagNumber_LeftTop=16#D012 AND DriveDiagNumber_RightTop=16#D012
			AND DriveDiagNumber_LeftBottom=16#D012 AND DriveDiagNumber_RightBottom=16#D012 THEN
			DriveStatus:=1;
		//D013, Axis state machine: Axis in operation
		ELSIF DriveDiagNumber_LeftTop=16#D013 AND DriveDiagNumber_RightTop=16#D013
			AND DriveDiagNumber_LeftBottom=16#D013 AND DriveDiagNumber_RightBottom=16#D013 THEN
			DriveStatus:=2;
		ELSE
			DriveStatus:=0;
		END_IF
	88:
		bDriveDiagMessageAndNumber:=FALSE;
		A_GetDriverStatusMC();
		GetDriveStatusStateDone:=TRUE;
		GetDriveStatusStateError:=FALSE;
		m_GetDriveStatusState:=0;
	-100:
		bDriveDiagMessageAndNumber:=FALSE;
		A_GetDriverStatusMC();
		GetDriveStatusStateDone:=FALSE;
		GetDriveStatusStateError:=TRUE;
		Error:=TRUE;
		ErrorId:=1301;
		ErrorDescription:='GetDriveStatusStateError';
END_CASE


(*IF bDriveDiagNumber THEN
    fbDriveDiagNumber_LeftTop(
       Axis     := LeftTopLin.NcToPlc,
       bExecute := TRUE,
       tTimeout := DEFAULT_ADS_TIMEOUT,
       iDiagNumber =>DriveDiagNumber_LeftTop
    );
    IF NOT fbDriveDiagNumber_LeftTop.bBusy THEN
        fbDriveDiagNumber_LeftTop(Axis := LeftTopLin.NcToPlc, bExecute := FALSE);
        bDriveDiagNumber := FALSE;
    END_IF
END_IF

IF bDriveDiagMessage THEN
    fbDriveDiagMessage_LeftTop(
       Axis     := LeftTopLin.NcToPlc,
       bExecute := TRUE,
       tTimeout := DEFAULT_ADS_TIMEOUT,
       sDiagMessage=>DriveDiagMessage_LeftTop
    );
    IF NOT fbDriveDiagMessage_LeftTop.bBusy THEN
        fbDriveDiagMessage_LeftTop(Axis := LeftTopLin.NcToPlc, bExecute := FALSE);
        bDriveDiagMessage := FALSE;
    END_IF
	DriveDiagMessageString_LeftTop:=DriveDiagMessage_LeftTop.strData;
END_IF
*)
END_ACTION

ACTION A_GetDriverStatusMC:
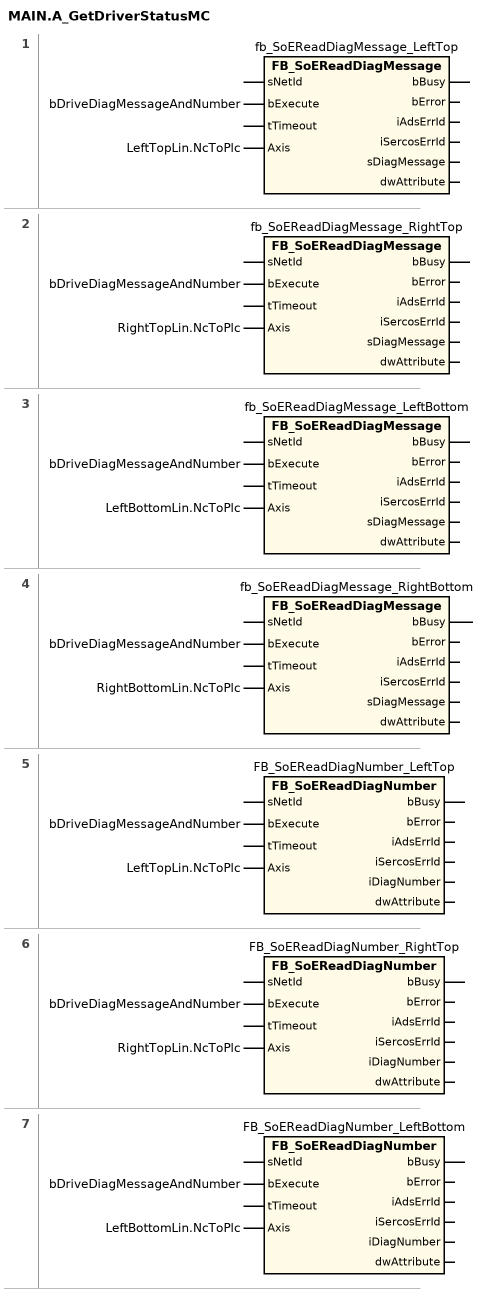
// NETWORK 1
fb_SoEReadDiagMessage_LeftTop(bExecute := bDriveDiagMessageAndNumber, Axis := LeftTopLin.NcToPlc); // FB_SoEReadDiagMessage

// NETWORK 2
fb_SoEReadDiagMessage_RightTop(bExecute := bDriveDiagMessageAndNumber, Axis := RightTopLin.NcToPlc); // FB_SoEReadDiagMessage

// NETWORK 3
fb_SoEReadDiagMessage_LeftBottom(bExecute := bDriveDiagMessageAndNumber, Axis := LeftBottomLin.NcToPlc); // FB_SoEReadDiagMessage

// NETWORK 4
fb_SoEReadDiagMessage_RightBottom(bExecute := bDriveDiagMessageAndNumber, Axis := RightBottomLin.NcToPlc); // FB_SoEReadDiagMessage

// NETWORK 5
FB_SoEReadDiagNumber_LeftTop(bExecute := bDriveDiagMessageAndNumber, Axis := LeftTopLin.NcToPlc); // FB_SoEReadDiagNumber

// NETWORK 6
FB_SoEReadDiagNumber_RightTop(bExecute := bDriveDiagMessageAndNumber, Axis := RightTopLin.NcToPlc); // FB_SoEReadDiagNumber

// NETWORK 7
FB_SoEReadDiagNumber_LeftBottom(bExecute := bDriveDiagMessageAndNumber, Axis := LeftBottomLin.NcToPlc); // FB_SoEReadDiagNumber

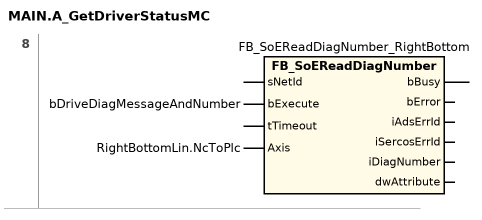
// NETWORK 8
FB_SoEReadDiagNumber_RightBottom(bExecute := bDriveDiagMessageAndNumber, Axis := RightBottomLin.NcToPlc); // FB_SoEReadDiagNumber
END_ACTION

ACTION A_GetTemperatureSensorsData:
//sensor_1
dut_sensor_datas_1.data_byte[3]:=Sensor_Reading_1[0];
dut_sensor_datas_1.data_byte[2]:=Sensor_Reading_1[1];
dut_sensor_datas_1.data_byte[1]:=Sensor_Reading_1[2];
dut_sensor_datas_1.data_byte[0]:=Sensor_Reading_1[3];
TemperatureSensors_1:=DINT_TO_LREAL(LREAL_TO_DINT(dut_sensor_datas_1.data_lreal*100))/100;
//sensor_2
dut_sensor_datas_2.data_byte[3]:=Sensor_Reading_2[0];
dut_sensor_datas_2.data_byte[2]:=Sensor_Reading_2[1];
dut_sensor_datas_2.data_byte[1]:=Sensor_Reading_2[2];
dut_sensor_datas_2.data_byte[0]:=Sensor_Reading_2[3];
TemperatureSensors_2:=DINT_TO_LREAL(LREAL_TO_DINT(dut_sensor_datas_2.data_lreal*100))/100;
//sensor_3
dut_sensor_datas_3.data_byte[3]:=Sensor_Reading_3[0];
dut_sensor_datas_3.data_byte[2]:=Sensor_Reading_3[1];
dut_sensor_datas_3.data_byte[1]:=Sensor_Reading_3[2];
dut_sensor_datas_3.data_byte[0]:=Sensor_Reading_3[3];
TemperatureSensors_3:=DINT_TO_LREAL(LREAL_TO_DINT(dut_sensor_datas_3.data_lreal*100))/100;
//sensor_4
dut_sensor_datas_4.data_byte[3]:=Sensor_Reading_4[0];
dut_sensor_datas_4.data_byte[2]:=Sensor_Reading_4[1];
dut_sensor_datas_4.data_byte[1]:=Sensor_Reading_4[2];
dut_sensor_datas_4.data_byte[0]:=Sensor_Reading_4[3];
TemperatureSensors_4:=DINT_TO_LREAL(LREAL_TO_DINT(dut_sensor_datas_4.data_lreal*100))/100;
//sensor_5
dut_sensor_datas_5.data_byte[3]:=Sensor_Reading_5[0];
dut_sensor_datas_5.data_byte[2]:=Sensor_Reading_5[1];
dut_sensor_datas_5.data_byte[1]:=Sensor_Reading_5[2];
dut_sensor_datas_5.data_byte[0]:=Sensor_Reading_5[3];
TemperatureSensors_5:=DINT_TO_LREAL(LREAL_TO_DINT(dut_sensor_datas_5.data_lreal*100))/100;
//sensor_6
dut_sensor_datas_6.data_byte[3]:=Sensor_Reading_6[0];
dut_sensor_datas_6.data_byte[2]:=Sensor_Reading_6[1];
dut_sensor_datas_6.data_byte[1]:=Sensor_Reading_6[2];
dut_sensor_datas_6.data_byte[0]:=Sensor_Reading_6[3];
TemperatureSensors_6:=DINT_TO_LREAL(LREAL_TO_DINT(dut_sensor_datas_6.data_lreal*100))/100;
//sensor_7
dut_sensor_datas_7.data_byte[3]:=Sensor_Reading_7[0];
dut_sensor_datas_7.data_byte[2]:=Sensor_Reading_7[1];
dut_sensor_datas_7.data_byte[1]:=Sensor_Reading_7[2];
dut_sensor_datas_7.data_byte[0]:=Sensor_Reading_7[3];
TemperatureSensors_7:=DINT_TO_LREAL(LREAL_TO_DINT(dut_sensor_datas_7.data_lreal*100))/100;
//sensor_8
dut_sensor_datas_8.data_byte[3]:=Sensor_Reading_8[0];
dut_sensor_datas_8.data_byte[2]:=Sensor_Reading_8[1];
dut_sensor_datas_8.data_byte[1]:=Sensor_Reading_8[2];
dut_sensor_datas_8.data_byte[0]:=Sensor_Reading_8[3];
TemperatureSensors_8:=DINT_TO_LREAL(LREAL_TO_DINT(dut_sensor_datas_8.data_lreal*100))/100;
//计算temperature_gradient
temperature_gradient_2_To_1:=ABS(TemperatureSensors_2-TemperatureSensors_1);
temperature_gradient_3_To_2:=ABS(TemperatureSensors_3-TemperatureSensors_2);
temperature_gradient_5_To_4:=ABS(TemperatureSensors_5-TemperatureSensors_4);
temperature_gradient_6_To_5:=ABS(TemperatureSensors_6-TemperatureSensors_5);
temperature_gradient_max:=DINT_TO_LREAL(LREAL_TO_DINT(MAX(temperature_gradient_2_To_1,temperature_gradient_3_To_2,
							temperature_gradient_5_To_4,temperature_gradient_6_To_5)*100))/100;
//计算大梁上的温度平均值
temperature_average:=DINT_TO_LREAL(LREAL_TO_DINT((TemperatureSensors_1+TemperatureSensors_2+TemperatureSensors_3+TemperatureSensors_4
					+TemperatureSensors_5+TemperatureSensors_6)/6*100))/100;
					

//传感器温度状态：0：有传感器度数错误；1:常温；2:低温；3:常温和低温中间态
IF TemperatureSensors_1=0 OR TemperatureSensors_2=0 OR TemperatureSensors_3=0 
	OR TemperatureSensors_4=0 OR TemperatureSensors_5=0 OR TemperatureSensors_6=0 THEN	
	temperatureStatus:=0;//有传感器读数错误
ELSIF TemperatureSensors_1>=RoomTemperatureThreshold AND TemperatureSensors_2>=RoomTemperatureThreshold AND TemperatureSensors_3>=RoomTemperatureThreshold
	AND TemperatureSensors_4>=RoomTemperatureThreshold AND TemperatureSensors_5>=RoomTemperatureThreshold AND TemperatureSensors_6>=RoomTemperatureThreshold THEN	
	temperatureStatus:=1;//常温
ELSIF TemperatureSensors_1<=CryogenicTemperatureThreshold AND TemperatureSensors_1>77
	AND TemperatureSensors_2<=CryogenicTemperatureThreshold  AND TemperatureSensors_2>77
	AND TemperatureSensors_3<=CryogenicTemperatureThreshold  AND TemperatureSensors_3>77
	AND TemperatureSensors_4<=CryogenicTemperatureThreshold   AND TemperatureSensors_4>77
	AND TemperatureSensors_5<=CryogenicTemperatureThreshold  AND TemperatureSensors_5>77
	AND TemperatureSensors_6<=CryogenicTemperatureThreshold   AND TemperatureSensors_6>77 THEN	
	temperatureStatus:=2;//低温
ELSE
	temperatureStatus:=3;//常温和低温中间
END_IF
END_ACTION

ACTION A_InitAxisParameters:
(*ÖáÎ»ÖÃ¡¢ËÙ¶È¡¢PosDiff*)

	Pos_LeftTopLin:=DINT_TO_LREAL(LREAL_TO_DINT(LeftTopLin.NcToPlc.ActPos*100000))/100000;
	Pos_RightTopLin:=DINT_TO_LREAL(LREAL_TO_DINT(RightTopLin.NcToPlc.ActPos*100000))/100000;
	Pos_LeftBottomLin:=DINT_TO_LREAL(LREAL_TO_DINT(LeftBottomLin.NcToPlc.ActPos*100000))/100000;
	Pos_RightBottomLin:=DINT_TO_LREAL(LREAL_TO_DINT(RightBottomLin.NcToPlc.ActPos*100000))/100000;

	
	LB_TestRecord:=Pos_LeftBottomLin-5;
	RB_TestRecord:=Pos_RightBottomLin-5;
	moveStatusLeftTop:=LeftTopLin.Status.Moving;
	moveStatusRightTop:=RightTopLin.Status.Moving;
	moveStatusLeftBottom:=LeftBottomLin.Status.Moving;
	moveStatusRightBottom:=RightBottomLin.Status.Moving;
	moveStatusAllAxis:=moveStatusLeftTop AND moveStatusRightTop AND moveStatusLeftBottom AND moveStatusRightBottom;

	Velo_LeftTopLin:=DINT_TO_LREAL(LREAL_TO_DINT(LeftTopLin.NcToPlc.ActVelo*100000))/100000;
	Velo_RightTopLin:=DINT_TO_LREAL(LREAL_TO_DINT(RightTopLin.NcToPlc.ActVelo*100000))/100000;
	Velo_LeftBottomLin:=DINT_TO_LREAL(LREAL_TO_DINT(LeftBottomLin.NcToPlc.ActVelo*100000))/100000;
	Velo_RightBottomLin:=DINT_TO_LREAL(LREAL_TO_DINT(RightBottomLin.NcToPlc.ActVelo*100000))/100000;

	PosDiff_LeftTopLin_actual:=LeftTopLin.NcToPlc.PosDiff;
	PosDiff_RightTopLin_actual:=RightTopLin.NcToPlc.PosDiff;
	PosDiff_LeftBottomLin_actual:=LeftBottomLin.NcToPlc.PosDiff;
	PosDiff_RightBottomLin_actual:=RightBottomLin.NcToPlc.PosDiff;

	LeftTopLin.ReadStatus();
	RightTopLin.ReadStatus();
	LeftBottomLin.ReadStatus();
	RightBottomLin.ReadStatus();
END_ACTION

ACTION A_InitRecipeParameters:
CASE state_loadParameters OF
	0:
		LoadParameter:=TRUE;
		Read_R_TRIG(CLK:=LoadParameter , Q=> );
		IF Read_R_TRIG.Q THEN
			state_loadParameters:=1;
		END_IF
	1:
		 ReturnDwordLoad:=RecipeManCommands.LoadAndWriteRecipe(RecipeDefinitionName:='Recipes' , RecipeName:='Parameters');
    	 LoadParameter:=FALSE;
		 IF ReturnDwordLoad<>0 THEN
		 	state_loadParameters:=-100;
		ELSE
			LoadRecipeParameters:=TRUE;
			LoadParameter:=FALSE;
			state_loadParameters:=88;
	 	END_IF
	88:
		loadParametersDone:=TRUE;
	-100:
		loadParametersDone:=FALSE;
		Error:=TRUE;
		ErrorId:=101;
		ErrorDescription:='LoadRecipeParameters Error';
		Plc_EmergencyStop:=FALSE;
END_CASE

////Save_R_TRIG(CLK:=SaveParameter , Q=> );
//Read_R_TRIG(CLK:=LoadParameter , Q=> );
//IF Save_R_TRIG.Q THEN  //将plc数据以文件形式保存在工控机中
//	 RecipeManCommands.CreateRecipe(RecipeDefinitionName:='Recipes' , RecipeName:='Parameters' );
//	 RecipeManCommands.ReadAndSaveRecipe(RecipeDefinitionName:='Recipes' , RecipeName:='Parameters' );
//	 SaveParameter:=FALSE;
//END_IF
//IF Read_R_TRIG.Q THEN  //将工控机中的文件数据读取到plc中
//     ReturnDwordLoad:=RecipeManCommands.LoadAndWriteRecipe(RecipeDefinitionName:='Recipes' , RecipeName:='Parameters');
//     LoadParameter:=FALSE;
//	 IF ReturnDwordLoad<>0 THEN
//		 Error:=TRUE;
//		 ErrorId:=101;
//		 ErrorDescription:='LoadRecipeParameters Error';
//		 Plc_EmergencyStop:=FALSE;
//	 END_IF
//END_IF
END_ACTION

ACTION A_KillOpcIocShellExe:
R_TRIG_Exekill(CLK:=bExe_Kill_Prog, Q=> );
CASE Exe_kill_step OF
	0:
		IF R_TRIG_Exekill.Q THEN
			NT_StartProcess_Kill.START:=FALSE;
			NT_StartProcess_Kill.PATHSTR:='C:\HZB\OpcIocShell\IDControlIOC\killcmd.bat';
			//NT_StartProcess_Kill.DIRNAME:='C:\Program Files (x86)\HZB\OpcIocShell\bin\opcIocShell.exe';
			Exe_kill_step:=10;
		END_IF;
	10:
		NT_StartProcess_Kill.START:=TRUE;
		Exe_kill_step:=20;
	20:
		IF NT_StartProcess_Kill.ERR THEN
			Exe_kill_step:=0;
		ELSE
			Exe_kill_step:=30;
		END_IF;

	30:
		NT_StartProcess_Kill.START:=TRUE;
		Exe_kill_step:=40;
	40:
		IF NOT NT_StartProcess_Kill.BUSY THEN
			NT_StartProcess_Kill.START:=FALSE;
			Exe_Kill_Done:=TRUE;
			Exe_kill_step:=0;
		END_IF;
END_CASE;

NT_StartProcess_Kill(
	NETID:='' ,
	PATHSTR:= ,
	DIRNAME:= , 
	COMNDLINE:= , 
	START:= ,
	ERRID=> );
END_ACTION

ACTION A_LoadOpcIocShellExe:
R_TRIG_Exeload(CLK:=bExe_load_Prog, Q=> );
LoadOpcIocTON(PT:=T#10S);
CASE Exe_load_step OF
	0:
		LoadOpcIocTON.IN:=TRUE;
		IF R_TRIG_Exeload.Q THEN
			NT_StartProcess_Load.START:=FALSE;
			NT_StartProcess_Load.PATHSTR:='C:\HZB\OpcIocShell\IDControlIOC\startTwinCATOPCServer.bat';
			Exe_load_step:=10;
		END_IF;
	10:
		IF LoadOpcIocTON.Q THEN
			NT_StartProcess_Load.START:=TRUE;
			Exe_load_step:=20;
		END_IF
	20:
		LoadOpcIocTON.IN:=FALSE;
		IF NT_StartProcess_Load.ERR THEN
			Exe_load_step:=0;
		ELSE
			Exe_load_step:=30;
		END_IF;
	30:
		IF NOT NT_StartProcess_Load.BUSY THEN
			NT_StartProcess_Load.START:=FALSE;
			Exe_Load_Done:=TRUE;
			Exe_load_step:=0;
		END_IF;
END_CASE;

NT_StartProcess_Load(
	NETID:='' ,
	PATHSTR:= ,
	DIRNAME:= , 
	COMNDLINE:= , 
	START:= ,
	ERRID=> );
END_ACTION

ACTION A_PosDiffDetectiion:
IF ABS(PosDiff_LeftTopLin_actual)>PosDiff_LeftTopLin THEN
	ErrorID:=201;
	Error:=TRUE;
	ErrorDescription:='ABS(PosDiff_LeftTopLin_actual)>PosDiff_LeftTopLin';
	FB_PlcEmergencyStop();
	LED_Error:=TRUE;
END_IF
IF ABS(PosDiff_RightTopLin_actual)>PosDiff_RightTopLin THEN
	ErrorID:=202;
	Error:=TRUE;
	ErrorDescription:='ABS(PosDiff_RightTopLin_actual)>PosDiff_RightTopLin';
	FB_PlcEmergencyStop();
	LED_Error:=TRUE;
END_IF
IF ABS(PosDiff_LeftBottomLin_actual)>PosDiff_LeftBottomLin THEN
	ErrorID:=203;
	Error:=TRUE;
	ErrorDescription:='ABS(PosDiff_LeftBottomLin_actual)>PosDiff_LeftBottomLin';
	FB_PlcEmergencyStop();
	LED_Error:=TRUE;
END_IF
IF ABS(PosDiff_RightBottomLin_actual)>PosDiff_RightBottomLin THEN
	ErrorID:=204;
	ErrorDescription:='ABS(PosDiff_RightBottomLin_actual)>PosDiff_RightBottomLin';
	Error:=TRUE;
	FB_PlcEmergencyStop();
	LED_Error:=TRUE;
END_IF
//
IF ABS(PosDiff_LeftTopLin_actual-PosDiff_RightTopLin_actual)>0.05 THEN
	ErrorID:=205;
	ErrorDescription:='ABS(PosDiff_LeftTopLin_actual-PosDiff_RightTopLin_actual)>0.05';
	Error:=TRUE;
	FB_PlcEmergencyStop();
	LED_Error:=TRUE;
ELSIF ABS(PosDiff_LeftBottomLin_actual-PosDiff_RightBottomLin_actual)>0.05 THEN
	ErrorID:=206;
	ErrorDescription:='ABS(PosDiff_LeftBottomLin_actual-PosDiff_RightBottomLin_actual)>0.05';
	Error:=TRUE;
	FB_PlcEmergencyStop();
	LED_Error:=TRUE;
END_IF
END_ACTION

ACTION A_RestartTC:
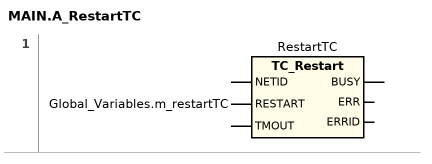
// NETWORK 1
RestartTC(RESTART := Global_Variables.m_restartTC); // TC_Restart
END_ACTION

ACTION A_SafePlcStartInit:
fb_ton0(PT:=t#1s);
fb_ton1(PT:=t#0.1s);
fb_ton2(PT:=t#0.1s);
fb_ton3(PT:=t#0.1s);

CASE SafeStatus OF
	0:
		IF COM_ERROR OR NOT Estop_Out THEN
			Err_Ack:=TRUE;
			fb_ton0.IN:=TRUE;
			SafeStatus:=1;
		ELSE
			SafePLCRunOK:=TRUE;
			SafeStatus:=0;
		END_IF
	1:
		IF fb_ton0.Q THEN
			Err_Ack:=FALSE;
			Safe_run:=TRUE;
			fb_ton1.IN:=TRUE;
			SafeStatus:=2;
		END_IF

	2:
		IF fb_ton1.Q THEN
			IF Estop_RunAndRestart=FALSE THEN
				Estop_RunAndRestart:=TRUE;
				fb_ton2.IN:=TRUE;
				SafeStatus:=3;
			END_IF
		END_IF
	3:
		IF fb_ton2.Q THEN
			IF Estop_RunAndRestart THEN
				Estop_RunAndRestart:=FALSE;
				fb_ton3.IN:=TRUE;
				SafeStatus:=4;
			END_IF
		END_IF
	4:
		IF fb_ton3.Q THEN
			IF Estop_Out THEN
				SafePLCRunOK:=TRUE;
				SafeStatus:=0;
			ELSE
				SafePLCRunOK:=FALSE;
				//Error:=TRUE;
				//ErrorId:=301;
				//ErrorDescription:='SafePLCRunOK fail';
			END_IF
		fb_ton0.IN:=FALSE;
		fb_ton1.IN:=FALSE;
		fb_ton2.IN:=FALSE;
		fb_ton3.IN:=FALSE;
		END_IF


END_CASE
END_ACTION

ACTION A_SetAxisPosition:
fb_ton4(PT:=t#0.5s);
CASE SetAxisPosState OF
	0:	(*FB_Set_AxisPosition*)
		FB_Set_AxisPosition(Execute:=TRUE);
		fb_ton4.IN:=TRUE;
		SetAxisPosState:=1;
	1:	(*wait*)
		FB_Set_AxisPosition();
		IF NOT FB_Set_AxisPosition.Done THEN		(*FB_Set_AxisPositionÃ»ÓÐÖ´ÐÐÍê£¬wait£¬³¬Ê±FB Error*)
			IF NOT fb_ton4.Q THEN
				SetAxisPosState:=1;
			ELSE
				SetAxisPosState:=99;
			END_IF
		ELSE
			SetAxisPosState:=88;
		END_IF
	88:
		SetAxisPosState:=0;
		SerAxisPositionDone:=TRUE;
		Error:=FALSE;
		ErrorID:=0;
		FB_Set_AxisPosition.Execute:=FALSE;
		fb_ton4.IN:=FALSE;
	99:
		SetAxisPosState:=99;
		SerAxisPositionDone:=FALSE;
		Error:=TRUE;
		FB_Set_AxisPosition.Execute:=FALSE;
		fb_ton4.IN:=FALSE;
		LED_Error:=TRUE;
		ErrorID:=401;
		ErrorDescription:='SetAxisPosition fail';
END_CASE
END_ACTION

ACTION A_SetLinearEncoderPositionBias:
//光栅positionBias补偿低温收缩量
IF CryogenicCompensationConditionsReady AND NOT CryogenicCompensationDone THEN
	PositionBias_LeftTop:=PositionBias_LeftTop+CryogenicCompensation_LeftTop;
	PositionBias_RightTop:=PositionBias_RightTop+CryogenicCompensation_RightTop;
	PositionBias_LeftBottom:=PositionBias_LeftBottom+CryogenicCompensation_LeftBottom;
	PositionBias_RightBottom:=PositionBias_RightBottom+CryogenicCompensation_RightBottom;
	CryogenicCompensationDone:=TRUE;
END_IF
//设置bias开始
A_SetLinearEncoderPositionBiasMC();
PositionBiasTON(PT:=T#0.1S);
CASE state_setLEPosBias OF
	0:
		PositionBiasTON.IN:=TRUE;
		IF MC_SetLEPosBias_LeftTop.Error OR MC_SetLEPosBias_RightTop.Error OR 
			MC_SetLEPosBias_LeftBottom.Error OR MC_SetLEPosBias_RightBottom.Error THEN
			state_setLEPosBias:=-100;
		ELSE 
			state_setLEPosBias:=1;
		END_IF
	1:
		IF NOT MC_SetLEPosBias_LeftTop.Done OR NOT MC_SetLEPosBias_RightTop.Done OR 
			NOT MC_SetLEPosBias_LeftBottom.Done OR NOT MC_SetLEPosBias_RightBottom.Done THEN
			MC_SetLEPosBias_LeftTop.Execute:=TRUE;
			MC_SetLEPosBias_RightTop.Execute:=TRUE;
			MC_SetLEPosBias_LeftBottom.Execute:=TRUE;
			MC_SetLEPosBias_RightBottom.Execute:=TRUE;
			state_setLEPosBias:=2;
		ELSE
			state_setLEPosBias:=-100;
		END_IF
	2:
		IF NOT MC_SetLEPosBias_LeftTop.Done OR NOT MC_SetLEPosBias_RightTop.Done OR 
			NOT MC_SetLEPosBias_LeftBottom.Done OR NOT MC_SetLEPosBias_RightBottom.Done THEN
			IF NOT PositionBiasTON.Q THEN
				state_setLEPosBias:=2;
			ELSE
				state_setLEPosBias:=-100;
			END_IF
		END_IF
		IF  MC_SetLEPosBias_LeftTop.Done AND MC_SetLEPosBias_RightTop.Done AND
			MC_SetLEPosBias_LeftBottom.Done AND MC_SetLEPosBias_RightBottom.Done THEN
			state_setLEPosBias:=88;
		END_IF	
		IF MC_SetLEPosBias_LeftTop.Error OR MC_SetLEPosBias_RightTop.Error OR 
			MC_SetLEPosBias_LeftBottom.Error OR MC_SetLEPosBias_RightBottom.Error THEN
			state_setLEPosBias:=-100;
		END_IF 
		
	88:
		PositionBiasTON.IN:=FALSE;
		PositionBiasDone:=TRUE;
	-100:
		PositionBiasTON.IN:=FALSE;
		PositionBiasDone:=FALSE;
		Error:=TRUE;
		ErrorId:=901;
		ErrorDescription:='Set LinearEncoderPositionBias Error';
		Plc_EmergencyStop:=FALSE;
END_CASE
END_ACTION

ACTION A_SetLinearEncoderPositionBiasMC:
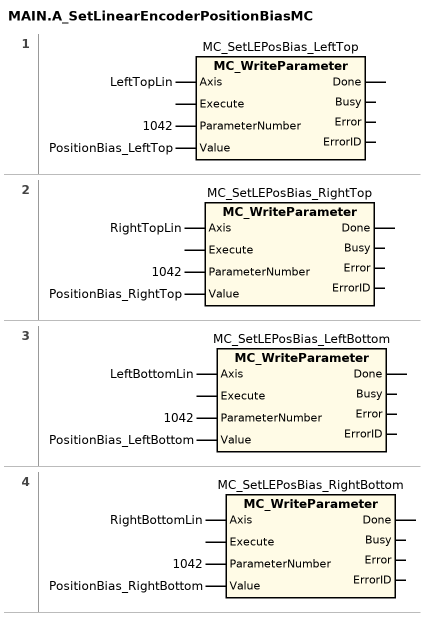
// NETWORK 1
MC_SetLEPosBias_LeftTop(Axis := LeftTopLin, ParameterNumber := 1042, Value := PositionBias_LeftTop); // MC_WriteParameter

// NETWORK 2
MC_SetLEPosBias_RightTop(Axis := RightTopLin, ParameterNumber := 1042, Value := PositionBias_RightTop); // MC_WriteParameter

// NETWORK 3
MC_SetLEPosBias_LeftBottom(Axis := LeftBottomLin, ParameterNumber := 1042, Value := PositionBias_LeftBottom); // MC_WriteParameter

// NETWORK 4
MC_SetLEPosBias_RightBottom(
    Axis := RightBottomLin,
    ParameterNumber := 1042,
    Value := PositionBias_RightBottom); // MC_WriteParameter
END_ACTION

END_PROGRAM

// ---- POUs/CommonFB/ExternFB/FB_LedShow.TcPOU
(****************************************************************
NAME:			FB_LedShow
DATA:			2017.2.16
VERSION:		1.0.0
DESCRIPTION:	FB_LedShow
HISTORY:
				2017.2.16 	NEW

***************************************************************)
FUNCTION_BLOCK FB_LedShow
VAR_INPUT
	Error:BOOL;
	Run:BOOL;
END_VAR
VAR_OUTPUT
	LedStatus:DINT;
END_VAR
VAR
END_VAR

IF Run THEN
	Led_Run:=TRUE;
	Led_Error:=FALSE;
	LedStatus:=1;
END_IF

IF Error THEN
	Led_Run:=FALSE;
	Led_Error:=TRUE;
	LedStatus:=0;
END_IF

END_FUNCTION_BLOCK

// ---- POUs/CommonFB/MainFB/FB_SetAxisPosition.TcPOU
(****************************************************************
NAME:			FB_SetAxisPosition
DATA:			2017.2.16
VERSION:		1.0.0
DESCRIPTION:	FB_SetAxisPosition
HISTORY:
				2017.2.16		NEW

***************************************************************)
FUNCTION_BLOCK FB_SetAxisPosition
VAR_INPUT
	//GapValueSet:LREAL:=0;
	ValueSet_LeftTop:LREAL:=0;
	ValueSet_RightTop:LREAL:=0;
	ValueSet_LeftBottom:LREAL:=0;
	ValueSet_RightBottom:LREAL:=0;
	Execute:BOOL;
END_VAR
VAR_OUTPUT
	FbID:DINT:=1001;
	State:DINT;
	Busy:BOOL;
	Done:BOOL;
	Error:BOOL;
	ErrorID:DINT;
END_VAR
VAR
	LeftTopLin_MC_SetPosition: MC_SetPosition;
	RightTopLin_MC_SetPosition: MC_SetPosition;
	LeftBottomLin_MC_SetPosition: MC_SetPosition;
	RightBottomLin_MC_SetPosition: MC_SetPosition;
	fb_ton: TON;
	FB_Couple_Axis: FB_CoupleAxis;
	FB_PlcEmergencyStop: FB_PlcEmergencyStop;
END_VAR

IF Execute THEN
Busy:=TRUE;
Done:=FALSE;
fb_ton(PT:=t#0.1s);
CASE State OF
	0:
		IF LeftTopLin_MC_SetPosition.Error OR RightTopLin_MC_SetPosition.Error
			OR LeftBottomLin_MC_SetPosition.Error OR RightBottomLin_MC_SetPosition.Error THEN		(*FB Error*)
			ErrorID:=1;
			State:=99;
		ELSIF FB_Couple_Axis.InGear THEN		(*²»ÄÜ³öÏÖÒÑ¾­ñîºÏÔÙÉèÖÃÎ»ÖÃµÄÇé¿ö£¬±ØÐëÏÈ½âñîºÏ£¬ÔÙÉèÖÃÎ»ÖÃ*)
			ErrorID:=2;
			State:=99;
		ELSIF LeftTopLin.NcToPlc.CoupleState=0 AND LeftBottomLin.NcToPlc.CoupleState=0
			AND RightTopLin.NcToPlc.CoupleState=0 AND RightBottomLin.NcToPlc.CoupleState=0 THEN	(*Öá¾ù´¦ÓÚÎÞñîºÏ×´Ì¬£¬¿ÉÒÔÉèÖÃÎ»ÖÃ£¬×ªÏÂÒ»²½*)
			State:=1;
		ELSE
			ErrorID:=3;
			State:=-100;
		END_IF
	1:	(*Execute*)
		LeftTopLin_MC_SetPosition.Position:=ValueSet_LeftTop;
		LeftTopLin_MC_SetPosition.Execute:=TRUE;
		RightTopLin_MC_SetPosition.Position:=ValueSet_RightTop;
		RightTopLin_MC_SetPosition.Execute:=TRUE;
		LeftBottomLin_MC_SetPosition.Position:=ValueSet_LeftBottom;
		LeftBottomLin_MC_SetPosition.Execute:=TRUE;
		RightBottomLin_MC_SetPosition.Position:=ValueSet_RightBottom;
		RightBottomLin_MC_SetPosition.Execute:=TRUE;
		A_SetPositionMC();
		fb_ton.IN:=TRUE;
		State:=2;
	2:	(*Wait*)
		A_SetPositionMC();
		IF NOT LeftTopLin_MC_SetPosition.Done OR NOT RightTopLin_MC_SetPosition.Done
			OR NOT LeftBottomLin_MC_SetPosition.Done OR NOT RightBottomLin_MC_SetPosition.Done THEN		(*DoneÐÅºÅ²»µ½£¬¼ÌÐøµÈ´ý£¬Èç¹û³¬Ê±ÔòFB Error*)
			IF NOT fb_ton.Q THEN
				State:=2;
			ELSE
				ErrorID:=4;
				State:=99;
			END_IF
		ELSIF  LeftTopLin_MC_SetPosition.Done AND RightTopLin_MC_SetPosition.Done
			AND LeftBottomLin_MC_SetPosition.Done AND RightBottomLin_MC_SetPosition.Done THEN		(*Done£¬×ªÏÂÒ»²½*)
			State:=88;
		ELSE
			ErrorID:=5;
			State:=99;
		END_IF
	88:
		Execute:=FALSE;
		State:=0;
		Busy:=FALSE;
		Done:=TRUE;
		Error:=FALSE;
		ErrorID:=0;
		LeftTopLin_MC_SetPosition.Execute:=FALSE;
		RightTopLin_MC_SetPosition.Execute:=FALSE;
		LeftBottomLin_MC_SetPosition.Execute:=FALSE;
		RightBottomLin_MC_SetPosition.Execute:=FALSE;
		fb_ton.IN:=FALSE;
	99:
		Execute:=FALSE;
		State:=99;
		Busy:=FALSE;
		Done:=FALSE;
		Error:=TRUE;
		LeftTopLin_MC_SetPosition.Execute:=FALSE;
		RightTopLin_MC_SetPosition.Execute:=FALSE;
		LeftBottomLin_MC_SetPosition.Execute:=FALSE;
		RightBottomLin_MC_SetPosition.Execute:=FALSE;
		fb_ton.IN:=FALSE;
	-100:
		FB_PlcEmergencyStop();
		Execute:=FALSE;
		State:=-100;
		Busy:=FALSE;
		Done:=FALSE;
		Error:=TRUE;
		LeftTopLin_MC_SetPosition.Execute:=FALSE;
		RightTopLin_MC_SetPosition.Execute:=FALSE;
		LeftBottomLin_MC_SetPosition.Execute:=FALSE;
		RightBottomLin_MC_SetPosition.Execute:=FALSE;
		fb_ton.IN:=FALSE;
END_CASE
END_IF

ACTION A_SetPositionMC:
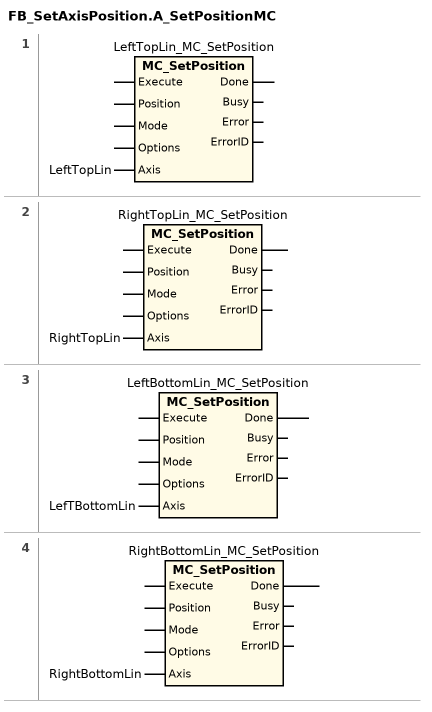
// NETWORK 1
LeftTopLin_MC_SetPosition(Axis := LeftTopLin); // MC_SetPosition

// NETWORK 2
RightTopLin_MC_SetPosition(Axis := RightTopLin); // MC_SetPosition

// NETWORK 3
LeftBottomLin_MC_SetPosition(Axis := LefTBottomLin); // MC_SetPosition

// NETWORK 4
RightBottomLin_MC_SetPosition(Axis := RightBottomLin); // MC_SetPosition
END_ACTION

END_FUNCTION_BLOCK

// ---- POUs/CommonFB/MainFB/FB_CoupleAxis.TcPOU
(****************************************************************
NAME:			FB_CoupleAxis
DATA:			2017.2.16
VERSION:		1.0.0
DESCRIPTION:	FB_CoupleAxis
HISTORY:
				2017.2.16		NEW

***************************************************************)
FUNCTION_BLOCK FB_CoupleAxis
VAR_INPUT
	Execute:BOOL;
	Reset:BOOL;
END_VAR
VAR_OUTPUT
	FbID:DINT:=1001;
	State:DINT;
	Busy:BOOL;
	InGear:BOOL;
	Error:BOOL;
	ErrorID:DINT;
END_VAR
VAR_IN_OUT
END_VAR
VAR
	Bottom_MC_GearIn: MC_GearIn;
	Top_MC_GearIn: MC_GearIn;
	fb_ton: TON;
END_VAR

IF Execute THEN
Busy:=TRUE;
InGear:=FALSE;
fb_ton(PT:=t#0.1s);
CASE State OF
	0:	(*Check*)
		IF LeftTopLin.NcToPlc.CoupleState=3 OR LeftBottomLin.NcToPlc.CoupleState=3 THEN	(*LeftTop»òÕßLeftBottomÎª´ÓÖá£¬Emergency Error*)
			ErrorID:=1;
			State:=-100;
		ELSIF LeftTopLin.NcToPlc.CoupleState=2 OR LeftBottomLin.NcToPlc.CoupleState=2
			OR RightTopLin.NcToPlc.CoupleState=2 OR RightBottomLin.NcToPlc.CoupleState=2 THEN	(*ÓÐÒ»ÖáCoupleStateÎª2£¬Emergency Error*)
			ErrorID:=2;
			State:=-100;
		ELSIF LeftTopLin.NcToPlc.CoupleState=1 AND LeftBottomLin.NcToPlc.CoupleState=1
			AND RightTopLin.NcToPlc.CoupleState=3 AND RightBottomLin.NcToPlc.CoupleState=3 THEN	(*ÒÑ¾­´¦ÓÚñîºÏ×´Ì¬*)
			ErrorID:=3;
			State:=-100;
		ELSIF LeftTopLin.Status.Moving OR  RightTopLin.Status.Moving OR LeftBottomLin.Status.Moving OR RightBottomLin.Status.Moving THEN	(*ÓÐÖáÔË¶¯*)
			ErrorID:=4;
			State:=-100;
		ELSIF  Top_MC_GearIn.Error OR Bottom_MC_GearIn.Error THEN		(*FB Error*)
			ErrorID:=5;
			State:=99;
		ELSIF Top_MC_GearIn.InGear OR Bottom_MC_GearIn.InGear THEN	(*ÒÑ¾­InGear£¬²»¿ÉÄÜ·¢Éú£¬FB Error*)
			ErrorID:=6;
			State:=99;
		ELSIF LeftTopLin.NcToPlc.CoupleState=0 AND LeftBottomLin.NcToPlc.CoupleState=0
			AND RightTopLin.NcToPlc.CoupleState=0 AND RightBottomLin.NcToPlc.CoupleState=0 THEN	(*Öá¾ù´¦ÓÚÎÞñîºÏ×´Ì¬£¬×ªÏÂÒ»²½*)
			State:=1;
		ELSE
			ErrorID:=7;
			State:=-100;
		END_IF
	1:	(*Couple*)
		IF LeftTopLin.NcToPlc.CoupleState=0 AND LeftBottomLin.NcToPlc.CoupleState=0
			AND RightTopLin.NcToPlc.CoupleState=0 AND RightBottomLin.NcToPlc.CoupleState=0 THEN	(*ÔÙ¼ì²é£¬Öá¾ù´¦ÓÚÎÞñîºÏ×´Ì¬£¬¿ªÊ¼ñîºÏ*)
			Top_MC_GearIn.Execute:=TRUE;
			Bottom_MC_GearIn.Execute:=TRUE;
			A_CoupleMC();
			fb_ton.IN:=TRUE;
			State:=2;
		ELSE
			ErrorID:=7;
			State:=99;
		END_IF
	2:	(*Couple Wait*)
		A_CoupleMC();
		IF NOT Top_MC_GearIn.InGear OR NOT Bottom_MC_GearIn.InGear THEN		(*InGearÐÅºÅ²»µ½£¬¼ÌÐøµÈ´ý£¬Èç¹û³¬Ê±ÔòFB Error*)
			IF NOT fb_ton.Q THEN
				State:=2;
			ELSE
				ErrorID:=8;
				State:=99;
			END_IF
		ELSIF  LeftTopLin.NcToPlc.CoupleState<>1 OR  RightTopLin.NcToPlc.CoupleState<>3
			OR LeftBottomLin.NcToPlc.CoupleState<>1 OR  RightBottomLin.NcToPlc.CoupleState<>3 THEN		(*ñîºÏ×´Ì¬²»¶Ô£¬Emergency Error*)
				ErrorID:=9;
				State:=-100;
		ELSIF   LeftTopLin.NcToPlc.CoupleState=1 AND  RightTopLin.NcToPlc.CoupleState=3
			AND LeftBottomLin.NcToPlc.CoupleState=1 AND  RightBottomLin.NcToPlc.CoupleState=3 THEN		(*ÕýÈ·ñîºÏ×´Ì¬£¬×ªÏÂÒ»²½*)
				State:=88;
		ELSE
				ErrorID:=10;
				State:=-100;
		END_IF
	88:	(*InGear*)
		Execute:=FALSE;
		State:=0;
		Busy:=FALSE;
		InGear:=TRUE;
		Error:=FALSE;
		ErrorID:=0;
		Bottom_MC_GearIn.Execute:=FALSE;
		Top_MC_GearIn.Execute:=FALSE;
		A_CoupleMC();
		fb_ton.IN:=FALSE;
	99:	(*FB Error*)
		Execute:=FALSE;
		State:=99;
		Busy:=FALSE;
		InGear:=FALSE;
		Error:=TRUE;
		Bottom_MC_GearIn.Execute:=FALSE;
		Top_MC_GearIn.Execute:=FALSE;
		A_CoupleMC();
		fb_ton.IN:=FALSE;
	-100:	(*Emergency Error*)
		FB_PlcEmergencyStop();
		Execute:=FALSE;
		State:=-100;
		Busy:=FALSE;
		InGear:=FALSE;
		Error:=TRUE;
		Bottom_MC_GearIn.Execute:=FALSE;
		Top_MC_GearIn.Execute:=FALSE;
		A_CoupleMC();
		fb_ton.IN:=FALSE;
END_CASE
END_IF
IF Reset THEN
		Execute:=FALSE;
		State:=0;
		Busy:=FALSE;
		InGear:=FALSE;
		Error:=FALSE;
		ErrorID:=0;
		Bottom_MC_GearIn.Execute:=FALSE;
		Top_MC_GearIn.Execute:=FALSE;
		A_CoupleMC();
		Reset:=FALSE;
END_IF

ACTION A_CoupleMC:
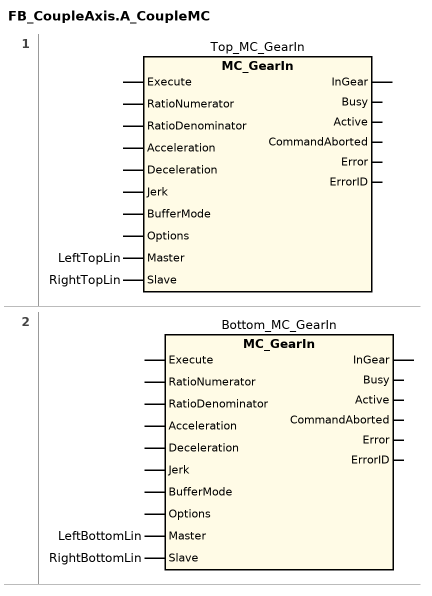
// NETWORK 1
Top_MC_GearIn(Master := LeftTopLin, Slave := RightTopLin); // MC_GearIn

// NETWORK 2
Bottom_MC_GearIn(Master := LeftBottomLin, Slave := RightBottomLin); // MC_GearIn
END_ACTION

END_FUNCTION_BLOCK

// ---- POUs/CommonFB/ExternFB/FB_PlcEmergencyStop.TcPOU
(****************************************************************
NAME:			FB_PlcEmergencyStop
DATA:			2017.2.15
VERSION:		1.0.0
DESCRIPTION:	PlcEmergencyStop
HISTORY:
				2017.2.15		NEW

***************************************************************)
FUNCTION_BLOCK FB_PlcEmergencyStop
VAR_INPUT
END_VAR
VAR_OUTPUT
	FbID:DINT:=2001;
	Busy:BOOL;
END_VAR
VAR
END_VAR

Plc_EmergencyStop:=FALSE;//FALSE is been triggered.
Busy:=TRUE;

END_FUNCTION_BLOCK

// ---- POUs/RS232/FB_SerialCom.TcPOU
FUNCTION_BLOCK FB_SerialCom
VAR_IN_OUT
	TxBuffer	: ComBuffer;
	RxBuffer	: ComBuffer;
END_VAR
VAR
	Timer		: TON := (PT:=T#1S);
	fbSend		: SendString;
	bSendBusy	: BOOL;
	eSendErrorID: ComError_t;

	fbReceive		: ReceiveString;
	sReceivedString	: STRING;
	sLastReceivedString: STRING;
	bStringReceived	: BOOL;
	bReceiveBusy	: BOOL;
	bReceiveError	: BOOL;
	eReceiveErrorID	: ComError_t;
	bReceiveTimeout	: BOOL;
	nReceiveCounter	: UDINT;
	sendErrorStatus: BOOL;
	RcvErrorStatus: BOOL;
	SendPreparedToString: STRING:='M0,0\r';
END_VAR

(* Call the send block every second TO REPEAT the transmission.
// Also call the block as long as it is busy to finish a transmission.*)
Timer(IN:=TRUE);
IF Timer.Q OR fbSend.Busy THEN
	Timer(IN:=FALSE); (* reset timer *)
	sendErrorStatus:=FALSE;
	fbSend(	SendString:= 'M0,0\r',
			TXbuffer:= TxBuffer,
			Busy=> bSendBusy,
			Error=> );
	IF fbSend.Error <> COMERROR_NOERROR THEN
		sendErrorStatus:=TRUE;
		eSendErrorID := fbSend.Error;
	END_IF
END_IF

(*//	Receive string data:
//	The block receives any data strings beginning with a STX ($02) and ending with an ETX ($03) character.	*)
fbReceive(
	Prefix:= '',
	Suffix:= '',
	Timeout:= T#1s,
	ReceivedString:= sReceivedString,
	RXbuffer:= RxBuffer,
	StringReceived=> bStringReceived,
	Busy=> bReceiveBusy,
	Error=> ,
	RxTimeout=> bReceiveTimeout );
IF fbReceive.Error <> COMERROR_NOERROR THEN
	RcvErrorStatus:=TRUE;
	eReceiveErrorID := fbReceive.Error;
ELSE
		RcvErrorStatus:=FALSE;
END_IF
IF bStringReceived THEN
	nReceiveCounter := nReceiveCounter + 1;
	sLastReceivedString := sReceivedString;
END_IF

END_FUNCTION_BLOCK

// ---- POUs/1.CarrierMode/SingleCarrierMode/SingleCarrierMode.TcPOU
PROGRAM SingleCarrierMode
VAR
	(*key Command*)
	btn_Power:BOOL;
	btn_PowerOn: BOOL;
	btn_PowerOff: BOOL;
	TopPositionNew:LREAL:=100;
	TopVelocityNew:LREAL:=1;
	btn_TopMove:BOOL;
	btn_TopStop:BOOL;
	BottomPositionNew:LREAL:=100;
	BottomVelocityNew:LREAL:=1;
	btn_BottomMove:BOOL;
	btn_BottomStop:BOOL;
	(*Var*)
	fb_ton1:TON;
	fb_ton2:TON;
	fb_ton3:TON;
	(*Status*)
	State:DINT;
	Busy:BOOL;
	TopBusy:BOOL;
	BottomBusy:BOOL;
	InitDone:BOOL;
	tm_state: DINT;
	ts_state: DINT;
	bm_state: DINT;
	bs_state: DINT;
	moni_State:DINT;
	(*PowerOff*)
	d_state: DINT;
	(*¼ì²âµ½ÏÞÎ»£¬»Ö¸´Move×´Ì¬*)
	FTrig_ReachLS: F_TRIG;
	FTrig_btn_GapMove: F_TRIG;
	InitPowerDone:BOOL;
END_VAR

TopPositionActual:=(Pos_LeftTopLin+Pos_RightTopLin)/2;
TopVelocityActual:=(Velo_LeftTopLin+Velo_RightTopLin)/2;
BottomPositionActual:=(Pos_LeftBottomLin+Pos_RightBOttomLin)/2;
BottomVelocityActual:=(Velo_LeftBottomLin+Velo_RightBOttomLin)/2;
(*btn_Power On/Off*)
IF btn_Power AND st_Power=0 THEN
	btn_PowerOn:=TRUE;
	btn_Power:=FALSE;
END_IF
IF btn_Power AND st_Power=1 THEN
	btn_PowerOff:=TRUE;
	btn_Power:=FALSE;
END_IF
IF btn_PowerOn THEN
	A_PowerOn();
END_IF
IF btn_PowerOff THEN
	A_PowerOff();
END_IF

(*********************************************************************Monitor All Carrirt Position***********************************************)
A_MonitoringAllAxis();
(*********************************************************************btn_TopMove*****************************************************************)
IF btn_TopMove AND NOT bottomBusy THEN
		TopBusy:=TRUE;
		btn_BottomMove:=FALSE;
		CASE tm_state OF
			0:
				FB_Move.Mode:=2;						(*单梁模式*)
				FB_Move.CoupleState:=st_Couple;			
				FB_Move.PowerState:=st_Power;			
				FB_Move.TopMove:=TRUE;				
				FB_Move.TopPosition:=TopPositionNew;		
				FB_Move.TopVelocity:=TopVelocityNew;		
				FB_Move();								
				tm_state:=1;
			1:
				FB_Move();
				LED_Run:=TRUE;
				IF NOT FB_Move.TopDone THEN	
					tm_state:=1;
				ELSE					
					tm_state:=88;
				END_IF
			88:
				btn_TopMove:=FALSE;	
				LED_Run:=FALSE;
				tm_state:=0;
				TopBusy:=FALSE;
		END_CASE
END_IF

(*********************************************************************btn_BottomMove*****************************************************************)
IF btn_BottomMove AND NOT TopBusy THEN
		btn_TopMove:=FALSE;
		BottomBusy:=TRUE;
		CASE bm_state OF
			0:
				FB_Move.Mode:=2;						
				FB_Move.CoupleState:=st_Couple;			
				FB_Move.PowerState:=st_Power;			
				FB_Move.BottomMove:=TRUE;			
				FB_Move.BottomPosition:=BottomPositionNew;		
				FB_Move.BottomVelocity:=BottomVelocityNew;		
				FB_Move();
				bm_state:=1;
			1:
				FB_Move();
				IF NOT FB_Move.BottomDone THEN
					LED_Run:=TRUE;
					bm_state:=1;
				ELSE
					bm_state:=88;
				END_IF
			88:
				BottomBusy:=FALSE;
				btn_TopMove:=FALSE;
				btn_BottomMove:=FALSE;
				bm_state:=0;
				LED_Run:=FALSE;
		END_CASE
END_IF
(*******************************************************************btn_TopStop********************************************************************)

IF btn_TopStop THEN
	LED_Run:=FALSE;
	TopMoveIndicator:=0;
	FB_Move.TopReset:=TRUE;
	TopBusy:=FALSE;
	FB_Move();
	btn_TopMove:=FALSE;	
	tm_state:=0;
	CASE ts_state OF
			0:
				FB_Stop.Mode:=2;
				FB_Stop.CoupleState:=st_Couple;
				FB_Stop.PowerState:=st_Power;
				FB_Stop.TopStop:=TRUE;	
				FB_Stop();	
				ts_state:=1;
			1:
				FB_Stop();
				IF NOT FB_Stop.TopDone THEN
					ts_state:=1;
				ELSE
					ts_state:=88;
				END_IF
			88:
				btn_TopStop:=FALSE;	
				FB_Move.TopReset:=FALSE;	
				ts_state:=0;
		END_CASE
END_IF
(*******************************************************************btn_BottomStop********************************************************************)
IF btn_BottomStop  THEN
	LED_Run:=FALSE;
	BottomMoveIndicator:=0;
	FB_Move.BottomReset:=TRUE;
	BottomBusy:=FALSE;
	FB_Move();			
	btn_BottomMove:=FALSE;			
	bm_state:=0;							
	CASE bs_state OF
			0:
				FB_Stop.Mode:=2;							
				FB_Stop.CoupleState:=st_Couple;			
				FB_Stop.PowerState:=st_Power;			
				FB_Stop.BottomStop:=TRUE;				
				FB_Stop();								
				bs_state:=1;
			1:
				FB_Stop();
				IF NOT FB_Stop.BottomDone THEN		
					bs_state:=1;
				ELSE									
					bs_state:=88;
				END_IF
			88:
				btn_BottomStop:=FALSE;					
				FB_Move.BottomReset:=FALSE;				
				bs_state:=0;
		END_CASE
END_IF
(*********************************************************************ÏÞÎ»Åö´¥×´Ì¬»Ö¸´************************************************************)

(*Èç¹û¼ì²âµ½ÏØÏÞÎ»¿ª¹ØÏÂ½µÑØ£¬»Ö¸´Move×´Ì¬*)
FTrig_ReachLS(CLK:=Unreach_LS_Top AND Unreach_LS_Bottom);
IF FTrig_ReachLS.Q THEN		(*FTrig_ReachLS.QÌ«¿ì£¬Ö»ÄÜÊ¹btn_TopStopÎªTRUE*)
	btn_TopStop:=TRUE;
	btn_BottomStop:=TRUE;
END_IF
IF btn_TopStop THEN			(*Òò´Ë£¬´Ë´¦Îªµ±Ö®Ç°btn_TopStopÎªTRUEÊ±£¬ÈËÎªÈÃbtn_BottomStopÎªTRUE*)
	btn_BottomStop:=TRUE;
END_IF
(*
(*Èç¹û¼ì²âµ½TopÏÞÎ»¿ª¹ØFALSE£¬ÇÒÄ¿±êÎ»ÖÃ´óÓÚµ±Ç°Î»ÖÃÊ±£¬»òÕßÏà·´Ê±£¬»Ö¸´Move×´Ì¬*)
IF NOT Unreach_LS_Top AND TopPositionNew-TopPositionActual>0.0005 AND btn_TopMove THEN
	btn_TopStop:=TRUE;
END_IF
IF NOT Unreach_LS_Bottom AND TopPositionNew-TopPositionActual<0.0005 AND btn_TopMove THEN
	btn_TopStop:=TRUE;
END_IF
IF NOT Unreach_LS_Top AND BottomPositionNew-BottomPositionActual>0.0005 AND btn_BottomMove THEN
	btn_BottomStop:=TRUE;
END_IF
IF NOT Unreach_LS_Bottom AND BottomPositionNew-BottomPositionActual<0.0005 AND btn_BottomMove THEN
	btn_BottomStop:=TRUE;
END_IF
*)

ACTION A_MonitoringAllAxis:
(****************************************************************
NAME:			A_MonitoringAllAxis
DATA:			2017.3.20
VERSION:		1.0.0
DESCRIPTION:	
				Ã¿´ÎÑ­»·¾ùÖ´ÐÐÖáÎ»ÖÃºÍÖáÔË¶¯µÄ¼ì²é
				1.4ÖáÏà¶ÔÔË¶¯¼ì²é
				2.4Öá¹âÕ¤³ßÎ»ÖÃ¡¢ËÙ¶È¶Ô±È¼ì²é
				3.Ã¿Öá¹âÕ¤ºÍ±àÂëÆ÷Î»ÖÃ¶Ô±È¼ì²é
HISTORY:
				2017.3.20		NEW

***************************************************************)
IF  st_Power<>0 THEN
		Diff_TopPos_actual:=Pos_leftTopLin-Pos_RightTopLin;
		Diff_TopVelo_actual:=Velo_leftTopLin-Velo_RightTopLin;
IF ABS(Pos_leftTopLin-Pos_RightTopLin)>Threshold_TopPos_SingleCarrier THEN
		btn_TopStop:=TRUE;
		btn_BottomStop:=TRUE;
		FB_PlcEmergencyStop();
		Error:=TRUE;
		ErrorID:=14;
		LED_Error:=TRUE;
ELSIF ABS(Velo_leftTopLin-Velo_RightTopLin)>Threshold_TopVelo_SingleCarrier  THEN
		(*btn_TopStop:=TRUE;
		btn_BottomStop:=TRUE;
		FB_PlcEmergencyStop();*)
		Error:=TRUE;
		ErrorID:=15;
(*Bottom Î»ÖÃºÍËÙ¶È±È¶Ô*)
ELSIF ABS(Pos_LeftBottomLin-Pos_RightBottomLin)>Threshold_BottomPos_SingleCarrier THEN
		btn_TopStop:=TRUE;
		btn_BottomStop:=TRUE;
		FB_PlcEmergencyStop();
		Error:=TRUE;
		ErrorID:=16;
		LED_Error:=TRUE;
ELSIF ABS(Velo_leftBottomLin-Velo_RightBottomLin)>Threshold_BottomVelo_SingleCarrier  THEN
		(*btn_TopStop:=TRUE;
		btn_BottomStop:=TRUE;
		FB_PlcEmergencyStop();*)
		Error:=TRUE;
		ErrorID:=17;
(*ÎÞLeftºÍRightËÙ¶ÈÎ»ÖÃµÄ¶Ô±È*)
END_IF
END_IF
(*********************************************************************************3.Ã¿Öá¹âÕ¤ºÍ±àÂëÆ÷Î»ÖÃ¶Ô±È¼ì²é**********************************************************************)
END_ACTION

ACTION A_PowerOff:
CASE d_state OF
		0:(*PowerOff*)
			FB_Power(Off:=TRUE);
				d_state:=1;
		1:
			IF NOT FB_power.OffStatus THEN
				d_state:=1;
			ELSE
				d_state:=88;
			END_IF
		88:(*ResetAllState*)
			btn_PowerOn:=FALSE;
			btn_TopMove:=FALSE;
			btn_TopStop:=FALSE;
			btn_BottomMove:=FALSE;
			btn_BottomStop:=FALSE;
			LeftTopLinMoveIndicator:=0;
			RightTopLinMoveIndicator:=0;
			LeftBottomLinMoveIndicator:=0;
			RightBottomLinMoveIndicator:=0;
			fb_ton1.IN:=FALSE;
			fb_ton2.IN:=FALSE;
			fb_ton3.IN:=FALSE;
			State:=0;
			Busy:=FALSE;
			InitPowerDone:=FALSE;
			Error:=FALSE;
			ErrorID:=0;
			tm_state:=0;
			ts_state:=0;
			bm_state:=0;
			bs_state:=0;
			btn_PowerOff:=FALSE;
			d_state:=0;
			Led_Run:=FALSE;
			Led_Error:=FALSE;
			moni_State:=0;
END_CASE
END_ACTION

ACTION A_PowerOn:
(****************************************************************
NAME:			A_PowerOn
DATA:			2018.1.9
VERSION:		1.0.0
DESCRIPTION:	
				ÉÏµãÃüÁîºó£¬Ë³ÐòÖ´ÐÐ£º
				1.FB_PowerOn
				·µ»ØÖ´ÐÐÊÇ·ñ³É¹¦
HISTORY:
				2019.1.9		NEW

***************************************************************)
fb_ton3(PT:=t#0.5s);
CASE State OF
	0:	(*FB_Power_On*)
		FB_Power(On:=TRUE);
		fb_ton3.IN:=TRUE;
		State:=1;
	1:	(*wait*)
		FB_power();
		IF NOT FB_power.OnStatus THEN		(*FB_Power_OnÃ»ÓÐÖ´ÐÐÍê£¬wait£¬³¬Ê±FB Error*)
			IF NOT fb_ton3.Q THEN
				State:=1;
			ELSE
				ErrorID:=1;
				State:=99;
			END_IF
		ELSE
			State:=88;
		END_IF
	88:	(*All Done*)
		btn_PowerOn:=FALSE;
		State:=0;
		Error:=FALSE;
		ErrorID:=0;
		Busy:=FALSE;
		InitPowerDone:=TRUE;
		FB_power.On:=FALSE;
		fb_ton3.IN:=FALSE;
		LED_Error:=FALSE;
	99:
		Error:=TRUE;
		//ErrorID:=701;
		//ErrorDescription:='power on error';		
		btn_PowerOn:=FALSE;
		State:=99;
		Busy:=FALSE;
		InitPowerDone:=FALSE;
		fb_ton3.IN:=FALSE;
		LED_Error:=TRUE;
END_CASE
END_ACTION

END_PROGRAM

// ---- POUs/CommonFB/MainFB/FB_Move.TcPOU
(****************************************************************
NAME:			FB_Move
DATA:			2017.2.17
VERSION:		1.0.0
DESCRIPTION:	FB_Move
HISTORY:
				2017.2.17		NEW
				2018.1.9		ÐÂÔöBCGapMode
***************************************************************)
FUNCTION_BLOCK FB_Move
VAR_INPUT
	(*È«¾Ö*)
	Mode:DINT;
	PowerState:BOOL;
	CoupleState:DINT;
	(*BCGapMode*)
	BCLeftTopPosition:LREAL;
	BCLeftTopVelocity:LREAL;
	BCRightTopPosition:LREAL;
	BCRightTopVelocity:LREAL;
	BCLeftBottomPosition:LREAL;
	BCLeftBottomVelocity:LREAL;
	BCRightBottomPosition:LREAL;
	BCRightBottomVelocity:LREAL;
	BCGapMove:BOOL;
	BCGapReset:BOOL;
	BCGapMove_2:BOOL;
	BCGapReset_2:BOOL;
	(*GapMode*)
	GapPosition:LREAL;
	GapVelocity:LREAL;
	GapMove:BOOL;
	GapReset:BOOL;
	(*SingleCarrierMode*)
	TopPosition:LREAL;
	TopVelocity:LREAL;
	TopMove:BOOL;
	TopReset:BOOL;
	BottomPosition:LREAL;
	BottomVelocity:LREAL;
	BottomMove:BOOL;
	BottomReset:BOOL;
	(*TaperMode*)
	TaperPosition:LREAL;
	TaperVelocity:LREAL;
	TaperMove:BOOL;
	TaperStop:BOOL;
	TaperReset:BOOL;
	(**DebugMode*)
	LeftTopPosition:LREAL;
	LeftTopVelocity:LREAL;
	LeftTopMove:BOOL;
	LeftTopStop:BOOL;
	LeftTopReset:BOOL;
	RightTopPosition:LREAL;
	RightTopVelocity:LREAL;
	RightTopMove:BOOL;
	RightTopStop:BOOL;
	RightTopReset:BOOL;
	LeftBottomPosition:LREAL;
	LeftBottomVelocity:LREAL;
	LeftBottomMove:BOOL;
	LeftBottomStop:BOOL;
	LeftBottomReset:BOOL;
	RightBottomPosition:LREAL;
	RightBottomVelocity:LREAL;
	RightBottomMove:BOOL;
	RightBottomStop:BOOL;
	RightBottomReset:BOOL;
END_VAR
VAR_OUTPUT
	FbID:DINT:=1001;
	GapState:DINT;
	GapBusy:BOOL;
	GapDone:BOOL;
	GapMoving:BOOL;

	BCGapState:DINT;
	BCGapBusy:BOOL;
	BCGapDone:BOOL;

	TopState:DINT;
	TopBusy:BOOL;
	TopDone:BOOL;
	BottomState:DINT;
	BottomBusy:BOOL;
	BottomDone:BOOL;

	TaperState:DINT;
	TaperBusy:BOOL;
	TaperDone:BOOL;

	LeftTopState:DINT;
	LeftTopBusy:BOOL;
	LeftTopDone:BOOL;
	RightTopState:DINT;
	RightTopBusy:BOOL;
	RightTopDone:BOOL;
	LeftBottomState:DINT;
	LeftBottomBusy:BOOL;
	LeftBottomDone:BOOL;
	RightBottomState:DINT;
	RightBottomBusy:BOOL;
	RightBottomDone:BOOL;


	Error:BOOL;
	ErrorID:DINT;
	
	GapState_2:DINT;
	GapBusy_2:BOOL;
	GapDone_2:BOOL;

	BCGapState_2:DINT;
	BCGapBusy_2:BOOL;
	BCGapDone_2:BOOL;
END_VAR
VAR
	Top_MC_MoveAbsolute: MC_MoveAbsolute;
	Bottom_MC_MoveAbsolute: MC_MoveAbsolute;
	RightTopLin_MC_MoveAbsolute: MC_MoveAbsolute;
	RightBottomLin_MC_MoveAbsolute: MC_MoveAbsolute;
	fb_ton: TON;
	fb_ton1: TON;
	fb_ton2: TON;
	fb_ton_debug_1:TON;
	fb_ton_debug_2:TON;
	fb_ton_debug_3:TON;
	fb_ton_debug_4:TON;
	fb_ton_BC:TON;
	fb_ton_BC_2:TON;
END_VAR

IF PowerState=1 THEN
	IF Mode=1 AND CoupleState=1 THEN
		A_GapMove();
	ELSIF Mode=2 AND CoupleState=0 AND TopMove THEN
		A_TopMove();
	ELSIF Mode=2 AND CoupleState=0 AND BottomMove THEN
		A_BottomMove();
	ELSIF Mode=3 AND CoupleState=0 AND TaperMove THEN
		A_TaperMove();
	ELSIF Mode=4 AND CoupleState=0 AND LeftTopMove THEN
		A_LeftTopMove();
	ELSIF Mode=4 AND CoupleState=0 AND RightTopMove THEN
		A_RightTopMove();
	ELSIF Mode=4 AND CoupleState=0 AND LeftBottomMove THEN
		A_LeftBottomMove();
	ELSIF Mode=4 AND CoupleState=0 AND RightBottomMove THEN
		A_RightBottomMove();
	ELSIF Mode=5 AND CoupleState=0 AND BCGapMove THEN
		A_BCGapMove();
	ELSIF Mode=6 AND CoupleState=0 AND BCGapMove_2 THEN
		A_BCGapMove_2();
	END_IF
END_IF

ACTION A_BCGapMove:
IF BCGapMove THEN
BCGapBusy:=TRUE;
BCGapDone:=FALSE;
fb_ton_BC(PT:=t#80s);(*2mm/s max spees,120mmÐÐ³Ì£¬60sÄÚ×ßÍê*)
(*×îºóÔÙ¼ì²éÒ»±éñîºÏ£¬²¹³¥Ä£Ê½ÏÂ£¬²»ÄÜñîºÏ*)
IF LeftTopLin.NcToPlc.CoupleState<>0 OR LeftBottomLin.NcToPlc.CoupleState<>0
			OR RightTopLin.NcToPlc.CoupleState<>0 OR RightBottomLin.NcToPlc.CoupleState<>0 THEN
			ErrorID:=1;
			GapState:=-100;
END_IF
A_MoveMC();
IF  LeftTopLin.Status.Moving AND RightTopLin.Status.Moving
			 AND LeftBottomLin.Status.Moving AND RightBottomLin.Status.Moving THEN
	GapMoving:=TRUE;
ELSE
	GapMoving:=FALSE;
END_IF
CASE BCGapState OF
	0:
		IF LeftTopLin.Status.Moving OR RightTopLin.Status.Moving
			 OR LeftBottomLin.Status.Moving OR RightBottomLin.Status.Moving THEN	(*ÖáÕýÔÚÔËÐÐ£¬Ñ­»·¸Ã²½µÈ´ý*)
			BCGapState:=88;
		ELSIF Top_MC_MoveAbsolute.Error OR Bottom_MC_MoveAbsolute.Error OR
				RightTopLin_MC_MoveAbsolute.Error OR RightBottomLin_MC_MoveAbsolute.Error THEN	(*¼ì²éMC Error*)
			ErrorID:=2;
			BCGapState:=99;
		(*ELSIF ABS(Pos_LeftTopLin-GapPosition/2)<0.002 AND  ABS(Pos_LeftBottomLin-GapPosition)<0.002 THEN	(*Ä¿±êÎ»ÖÃÓëµ±Ç°Î»ÖÃÒ»Ñù£¬²»¶¯*)
			GapState:=88;*)
		ELSIF leftTopLin.Status.NotMoving AND  leftBottomLin.Status.NotMoving
			 AND RightTopLin.Status.NotMoving AND RightBottomLin.Status.NotMoving THEN	(*Öá¶¼´¦ÓÚÍ£Ö¹×´Ì¬Ê±£¬×ªÏÂÒ»²½*)
			BCGapState:=1;
		END_IF
	1:
		Top_MC_MoveAbsolute.Position:=BCLeftTopPosition;
		Top_MC_MoveAbsolute.Velocity:=BCLeftTopVelocity;
		Bottom_MC_MoveAbsolute.Position:=BCLeftBottomPosition;
		Bottom_MC_MoveAbsolute.Velocity:=BCLeftBottomVelocity;
		RightTopLin_MC_MoveAbsolute.Position:=BCRightTopPosition;
		RightTopLin_MC_MoveAbsolute.Velocity:=BCRightTopVelocity;
		RightBottomLin_MC_MoveAbsolute.Position:=BCRightBottomPosition;
		RightBottomLin_MC_MoveAbsolute.Velocity:=BCRightBottomVelocity;
		Top_MC_MoveAbsolute.Execute:=TRUE;
		Bottom_MC_MoveAbsolute.Execute:=TRUE;
		RightTopLin_MC_MoveAbsolute.Execute:=TRUE;
		RightBottomLin_MC_MoveAbsolute.Execute:=TRUE;
		fb_ton_BC.IN:=TRUE;
		BCGapState:=2;
	2:
		IF NOT Top_MC_MoveAbsolute.Done OR NOT  Bottom_MC_MoveAbsolute.Done
				OR NOT RightTopLin_MC_MoveAbsolute.Done OR NOT RightBottomLin_MC_MoveAbsolute.Done THEN		(*ÔË¶¯ÖÐ£¬¼ì²éDoneÐÅºÅ£¬Ã»ÓÐÔòÑ­»·*)
			BCGapState:=2;
		ELSIF Top_MC_MoveAbsolute.Done  AND  Bottom_MC_MoveAbsolute.Done AND RightTopLin_MC_MoveAbsolute.Done AND RightBottomLin_MC_MoveAbsolute.Done THEN		(*ÔË¶¯Íê³É£¬×ªÏÂÒ»²½*)
			BCGapState:=88;
		END_IF
		(*½ÓÊÕµ½stopÐÅºÅÊ±£¬reset×´Ì¬*)
		IF BCGapReset THEN
			BCGapState:=89;
		END_IF

	88:
		BCGapMove:=FALSE;
		BCGapState:=0;
		BCGapBusy:=FALSE;
		BCGapDone:=TRUE;
		Error:=FALSE;
		ErrorID:=0;
		Top_MC_MoveAbsolute.Execute:=FALSE;
		Bottom_MC_MoveAbsolute.Execute:=FALSE;
		RightTopLin_MC_MoveAbsolute.Execute:=FALSE;
		RightBottomLin_MC_MoveAbsolute.Execute:=FALSE;
		fb_ton_BC.IN:=FALSE;
	89:
		BCGapMove:=FALSE;
		BCGapState:=0;
		BCGapBusy:=FALSE;
		BCGapDone:=FALSE;
		Error:=FALSE;
		ErrorID:=0;
		Top_MC_MoveAbsolute.Execute:=FALSE;
		Bottom_MC_MoveAbsolute.Execute:=FALSE;
		RightTopLin_MC_MoveAbsolute.Execute:=FALSE;
		RightBottomLin_MC_MoveAbsolute.Execute:=FALSE;
		fb_ton_BC.IN:=FALSE;
	99:
		BCGapMove:=FALSE;
		BCGapState:=99;
		BCGapBusy:=FALSE;
		BCGapDone:=FALSE;
		Error:=TRUE;
		Top_MC_MoveAbsolute.Execute:=FALSE;
		Bottom_MC_MoveAbsolute.Execute:=FALSE;
		RightTopLin_MC_MoveAbsolute.Execute:=FALSE;
		RightBottomLin_MC_MoveAbsolute.Execute:=FALSE;
		fb_ton_BC.IN:=FALSE;
	-100:
		FB_PlcEmergencyStop();
		BCGapMove:=FALSE;
		BCGapState:=-100;
		BCGapBusy:=FALSE;
		BCGapDone:=FALSE;
		Error:=TRUE;
		Top_MC_MoveAbsolute.Execute:=FALSE;
		Bottom_MC_MoveAbsolute.Execute:=FALSE;
		RightTopLin_MC_MoveAbsolute.Execute:=FALSE;
		RightBottomLin_MC_MoveAbsolute.Execute:=FALSE;
		fb_ton_BC.IN:=FALSE;
END_CASE
END_IF
END_ACTION

ACTION A_BCGapMove_2:
IF BCGapMove_2 THEN
BCGapBusy_2:=TRUE;
BCGapDone_2:=FALSE;
fb_ton_BC_2(PT:=T#80S);(*2mm/s max spees,120mmÐÐ³Ì£¬60sÄÚ×ßÍê*)
(*×îºóÔÙ¼ì²éÒ»±éñîºÏ£¬²¹³¥Ä£Ê½ÏÂ£¬²»ÄÜñîºÏ*)
IF LeftTopLin.NcToPlc.CoupleState<>0 OR LeftBottomLin.NcToPlc.CoupleState<>0
			OR RightTopLin.NcToPlc.CoupleState<>0 OR RightBottomLin.NcToPlc.CoupleState<>0 THEN
			ErrorID:=1;
			GapState:=-100;
END_IF
A_MoveMC();
CASE BCGapState_2 OF
	0:
		IF LeftTopLin.Status.Moving OR RightTopLin.Status.Moving
			 OR LeftBottomLin.Status.Moving OR RightBottomLin.Status.Moving THEN	(*ÖáÕýÔÚÔËÐÐ£¬Ñ­»·¸Ã²½µÈ´ý*)
			BCGapState_2:=88;
		ELSIF Top_MC_MoveAbsolute.Error OR Bottom_MC_MoveAbsolute.Error OR
				RightTopLin_MC_MoveAbsolute.Error OR RightBottomLin_MC_MoveAbsolute.Error THEN	(*¼ì²éMC Error*)
			ErrorID:=2;
			BCGapState_2:=99;
		(*ELSIF ABS(Pos_LeftTopLin-GapPosition/2)<0.002 AND  ABS(Pos_LeftBottomLin-GapPosition)<0.002 THEN	(*Ä¿±êÎ»ÖÃÓëµ±Ç°Î»ÖÃÒ»Ñù£¬²»¶¯*)
			GapState:=88;*)
		ELSIF leftTopLin.Status.NotMoving AND  leftBottomLin.Status.NotMoving
			 AND RightTopLin.Status.NotMoving AND RightBottomLin.Status.NotMoving THEN	(*Öá¶¼´¦ÓÚÍ£Ö¹×´Ì¬Ê±£¬×ªÏÂÒ»²½*)
			BCGapState_2:=1;
		END_IF
	1:
		Top_MC_MoveAbsolute.Position:=BCLeftTopPosition;
		Top_MC_MoveAbsolute.Velocity:=BCLeftTopVelocity;
		Bottom_MC_MoveAbsolute.Position:=BCLeftBottomPosition;
		Bottom_MC_MoveAbsolute.Velocity:=BCLeftBottomVelocity;
		RightTopLin_MC_MoveAbsolute.Position:=BCRightTopPosition;
		RightTopLin_MC_MoveAbsolute.Velocity:=BCRightTopVelocity;
		RightBottomLin_MC_MoveAbsolute.Position:=BCRightBottomPosition;
		RightBottomLin_MC_MoveAbsolute.Velocity:=BCRightBottomVelocity;
		Top_MC_MoveAbsolute.Execute:=TRUE;
		Bottom_MC_MoveAbsolute.Execute:=TRUE;
		RightTopLin_MC_MoveAbsolute.Execute:=TRUE;
		RightBottomLin_MC_MoveAbsolute.Execute:=TRUE;
		fb_ton_BC_2.IN:=TRUE;
		BCGapState_2:=2;
	2:
		IF NOT Top_MC_MoveAbsolute.Done OR NOT  Bottom_MC_MoveAbsolute.Done
				OR NOT RightTopLin_MC_MoveAbsolute.Done OR NOT RightBottomLin_MC_MoveAbsolute.Done THEN		(*ÔË¶¯ÖÐ£¬¼ì²éDoneÐÅºÅ£¬Ã»ÓÐÔòÑ­»·*)
			BCGapState_2:=2;
		ELSIF Top_MC_MoveAbsolute.Done  AND  Bottom_MC_MoveAbsolute.Done AND RightTopLin_MC_MoveAbsolute.Done AND RightBottomLin_MC_MoveAbsolute.Done THEN		(*ÔË¶¯Íê³É£¬×ªÏÂÒ»²½*)
			BCGapState_2:=88;
		END_IF
		(*½ÓÊÕµ½stopÐÅºÅÊ±£¬reset×´Ì¬*)
		IF BCGapReset_2 THEN
			BCGapState_2:=89;
		END_IF

	88:
		BCGapMove_2:=FALSE;
		BCGapState_2:=0;
		BCGapBusy_2:=FALSE;
		BCGapDone_2:=TRUE;
		Error:=FALSE;
		ErrorID:=0;
		Top_MC_MoveAbsolute.Execute:=FALSE;
		Bottom_MC_MoveAbsolute.Execute:=FALSE;
		RightTopLin_MC_MoveAbsolute.Execute:=FALSE;
		RightBottomLin_MC_MoveAbsolute.Execute:=FALSE;
		fb_ton_BC_2.IN:=FALSE;
	89:
		BCGapMove_2:=FALSE;
		BCGapState_2:=0;
		BCGapBusy_2:=FALSE;
		BCGapDone_2:=FALSE;
		Error:=FALSE;
		ErrorID:=0;
		Top_MC_MoveAbsolute.Execute:=FALSE;
		Bottom_MC_MoveAbsolute.Execute:=FALSE;
		RightTopLin_MC_MoveAbsolute.Execute:=FALSE;
		RightBottomLin_MC_MoveAbsolute.Execute:=FALSE;
		fb_ton_BC_2.IN:=FALSE;
	99:
		BCGapMove_2:=FALSE;
		BCGapState_2:=99;
		BCGapBusy_2:=FALSE;
		BCGapDone_2:=FALSE;
		Error:=TRUE;
		Top_MC_MoveAbsolute.Execute:=FALSE;
		Bottom_MC_MoveAbsolute.Execute:=FALSE;
		RightTopLin_MC_MoveAbsolute.Execute:=FALSE;
		RightBottomLin_MC_MoveAbsolute.Execute:=FALSE;
		fb_ton_BC_2.IN:=FALSE;
	-100:
		FB_PlcEmergencyStop();
		BCGapMove_2:=FALSE;
		BCGapState_2:=-100;
		BCGapBusy_2:=FALSE;
		BCGapDone_2:=FALSE;
		Error:=TRUE;
		Top_MC_MoveAbsolute.Execute:=FALSE;
		Bottom_MC_MoveAbsolute.Execute:=FALSE;
		RightTopLin_MC_MoveAbsolute.Execute:=FALSE;
		RightBottomLin_MC_MoveAbsolute.Execute:=FALSE;
		fb_ton_BC_2.IN:=FALSE;
END_CASE
END_IF
END_ACTION

ACTION A_BottomMove:
IF BottomMove THEN
BottomBusy:=TRUE;
BottomDone:=FALSE;
fb_ton2(PT:=t#80s);(*2mm/s max spees,120mmÐÐ³Ì£¬60sÄÚ×ßÍê*)
A_MoveMC();
CASE BottomState OF

	0:
		IF LeftTopLin.Status.Moving OR RightTopLin.Status.Moving
			 OR LeftBottomLin.Status.Moving OR RightBottomLin.Status.Moving THEN	(*ÖáÕýÔÚÔËÐÐ£¬Ñ­»·¸Ã²½µÈ´ý*)
			TopState:=88;
		ELSIF  Bottom_MC_MoveAbsolute.Error OR RightBottomLin_MC_MoveAbsolute.Error THEN		(*¼ì²éMC Error*)
			ErrorID:=2;
			BottomState:=99;
		ELSIF leftTopLin.Status.NotMoving AND  leftBottomLin.Status.NotMoving
			 AND RightTopLin.Status.NotMoving AND RightBottomLin.Status.NotMoving THEN	(*Öá¶¼´¦ÓÚÍ£Ö¹×´Ì¬Ê±£¬×ªÏÂÒ»²½*)
			BottomState:=1;
		END_IF
	1:
		Bottom_MC_MoveAbsolute.Position:=BottomPosition;
		Bottom_MC_MoveAbsolute.Velocity:=BottomVelocity;
		Bottom_MC_MoveAbsolute.Execute:=TRUE;
		RightBottomLin_MC_MoveAbsolute.Position:=BottomPosition;
		RightBottomLin_MC_MoveAbsolute.Velocity:=BottomVelocity;
		RightBottomLin_MC_MoveAbsolute.Execute:=TRUE;
		fb_ton2.IN:=TRUE;
		BottomState:=2;
	2:
		IF leftTopLin.Status.Moving OR RightTopLin.Status.Moving THEN	(*ÉÏÁº¶¯,ESTOP*)
			ErrorID:=3;
			BottomState:=-100;
		ELSIF  (LeftBottomLin.Status.Moving AND  RightBottomLin.Status.NotMoving)
				OR (RightBottomLin.Status.Moving AND  LeftBottomLin.Status.NotMoving) THEN
			ErrorID:=4;
			BottomState:=-100;
		ELSIF NOT Bottom_MC_MoveAbsolute.Done THEN		(*ÔË¶¯ÖÐ£¬¼ì²éDoneÐÅºÅ£¬Ã»ÓÐÔòÑ­»·£¬³¬Ê±±¨´í*)
			BottomState:=2;
		ELSIF Bottom_MC_MoveAbsolute.Done THEN		(*ÔË¶¯Íê³É£¬×ªÏÂÒ»²½*)
				BottomState:=88;
		END_IF
		(*½ÓÊÕµ½stopÐÅºÅÊ±£¬reset×´Ì¬*)
		IF BottomReset THEN
			BottomState:=89;
		END_IF

	88:
		BottomMove:=FALSE;
		BottomState:=0;
		BottomBusy:=FALSE;
		BottomDone:=TRUE;
		Error:=FALSE;
		ErrorID:=0;
		Bottom_MC_MoveAbsolute.Execute:=FALSE;
		RightBottomLin_MC_MoveAbsolute.Execute:=FALSE;
		fb_ton2.IN:=FALSE;
	89:
		BottomMove:=FALSE;
		BottomState:=0;
		BottomBusy:=FALSE;
		BottomDone:=FALSE;
		Error:=FALSE;
		ErrorID:=0;
		Bottom_MC_MoveAbsolute.Execute:=FALSE;
		RightBottomLin_MC_MoveAbsolute.Execute:=FALSE;
		fb_ton2.IN:=FALSE;
	99:
		BottomMove:=FALSE;
		BottomState:=99;
		BottomBusy:=FALSE;
		BottomDone:=FALSE;
		Error:=TRUE;
		Bottom_MC_MoveAbsolute.Execute:=FALSE;
		RightBottomLin_MC_MoveAbsolute.Execute:=FALSE;
		fb_ton2.IN:=FALSE;
	-100:
		FB_PlcEmergencyStop();
		BottomMove:=FALSE;
		BottomState:=-100;
		BottomBusy:=FALSE;
		BottomDone:=FALSE;
		Error:=TRUE;
		Bottom_MC_MoveAbsolute.Execute:=FALSE;
		RightBottomLin_MC_MoveAbsolute.Execute:=FALSE;
		fb_ton2.IN:=FALSE;
END_CASE
END_IF
END_ACTION

ACTION A_GapMove:
IF GapMove THEN
GapBusy:=TRUE;
GapDone:=FALSE;
fb_ton(PT:=t#80s);(*2mm/s max spees,120mmÐÐ³Ì£¬60sÄÚ×ßÍê*)
(*×îºóÔÙ¼ì²éÒ»±éñîºÏ*)
IF LeftTopLin.NcToPlc.CoupleState<>1 OR LeftBottomLin.NcToPlc.CoupleState<>1
			OR RightTopLin.NcToPlc.CoupleState<>3 OR RightBottomLin.NcToPlc.CoupleState<>3 THEN
			ErrorID:=1;
			GapState:=-100;
END_IF
A_MoveMC();
CASE GapState OF

	0:
		IF LeftTopLin.Status.Moving OR RightTopLin.Status.Moving
			 OR LeftBottomLin.Status.Moving OR RightBottomLin.Status.Moving THEN	(*ÖáÕýÔÚÔËÐÐ£¬Ñ­»·¸Ã²½µÈ´ý*)
			GapState:=88;
		ELSIF Top_MC_MoveAbsolute.Error OR Bottom_MC_MoveAbsolute.Error THEN		(*¼ì²éMC Error*)
			ErrorID:=2;
			GapState:=99;
		ELSIF ABS(Pos_LeftTopLin-GapPosition/2)<0.002 AND  ABS(Pos_LeftBottomLin-GapPosition)<0.002 THEN	(*Ä¿±êÎ»ÖÃÓëµ±Ç°Î»ÖÃÒ»Ñù£¬²»¶¯*)
			GapState:=88;
		ELSIF leftTopLin.Status.NotMoving AND  leftBottomLin.Status.NotMoving
			 AND RightTopLin.Status.NotMoving AND RightBottomLin.Status.NotMoving THEN	(*Öá¶¼´¦ÓÚÍ£Ö¹×´Ì¬Ê±£¬×ªÏÂÒ»²½*)
			GapState:=1;
		END_IF
	1:
		Top_MC_MoveAbsolute.Position:=GapPosition/2;
		Top_MC_MoveAbsolute.Velocity:=GapVelocity/2;
		Bottom_MC_MoveAbsolute.Position:=GapPosition/2;
		Bottom_MC_MoveAbsolute.Velocity:=GapVelocity/2;
		Top_MC_MoveAbsolute.Execute:=TRUE;
		Bottom_MC_MoveAbsolute.Execute:=TRUE;
		fb_ton.IN:=TRUE;
		GapState:=2;
	2:
		(*IF leftTopLin.Status.Moving AND   leftBottomLin.Status.NotMoving THEN (*ÉÏÏÂÁº²»Í¬Ê±¶¯*)
			ErrorID:=3;
			GapState:=-100;
		ELSIF RightTopLin.Status.NotMoving AND RightBottomLin.Status.Moving THEN (*ÉÏÏÂÁº²»Í¬Ê±¶¯*)
			ErrorID:=4;
			GapState:=-100;
		*)
		IF  (LeftTopLin.Status.Moving AND  RightTopLin.Status.NotMoving)
			OR  (LeftTopLin.Status.Moving AND LeftBottomLin.Status.NotMoving)
			OR (LeftTopLin.Status.Moving AND  RightBottomLin.Status.NotMoving)
				OR (RightTopLin.Status.Moving AND  LeftTopLin.Status.NotMoving)
				OR (RightTopLin.Status.Moving AND  LeftBottomLin.Status.NotMoving)
				OR (RightTopLin.Status.Moving AND  RightBottomLin.Status.NotMoving)
					OR (LeftBottomLin.Status.Moving AND  LeftTopLin.Status.NotMoving)
					OR (LeftBottomLin.Status.Moving AND  RightTopLin.Status.NotMoving)
					OR (LeftBottomLin.Status.Moving AND  RightBottomLin.Status.NotMoving)
						OR (RightBottomLin.Status.Moving AND  LeftTopLin.Status.NotMoving)
						OR (RightBottomLin.Status.Moving AND  RightTopLin.Status.NotMoving)
						OR (RightBottomLin.Status.Moving AND  LeftBottomLin.Status.NotMoving) THEN			(*Ò»Öá¶¯£¬ÆäËüÖá²»¶¯£¬½ô¼±×´Ì¬*)
			ErrorID:=5;
			GapState:=-100;
		ELSIF NOT Top_MC_MoveAbsolute.Done OR NOT  Bottom_MC_MoveAbsolute.Done THEN		(*ÔË¶¯ÖÐ£¬¼ì²éDoneÐÅºÅ£¬Ã»ÓÐÔòÑ­»·£¬³¬Ê±±¨´í*)
			(*IF NOT  fb_ton.Q THEN
				GapState:=2;
			ELSE
				ErrorID:=5;
				GapState:=-100;
			END_IF*)
			GapState:=2;
		ELSIF Top_MC_MoveAbsolute.Done  AND  Bottom_MC_MoveAbsolute.Done THEN		(*ÔË¶¯Íê³É£¬×ªÏÂÒ»²½*)
				GapState:=88;
		END_IF
		(*½ÓÊÕµ½stopÐÅºÅÊ±£¬reset×´Ì¬*)
		IF GapReset THEN
			GapState:=89;
		END_IF

	88:
		GapMove:=FALSE;
		GapState:=0;
		GapBusy:=FALSE;
		GapDone:=TRUE;
		Error:=FALSE;
		ErrorID:=0;
		Top_MC_MoveAbsolute.Execute:=FALSE;
		Bottom_MC_MoveAbsolute.Execute:=FALSE;
		fb_ton.IN:=FALSE;
	89:
		GapMove:=FALSE;
		GapState:=0;
		GapBusy:=FALSE;
		GapDone:=FALSE;
		Error:=FALSE;
		ErrorID:=0;
		Top_MC_MoveAbsolute.Execute:=FALSE;
		Bottom_MC_MoveAbsolute.Execute:=FALSE;
		fb_ton.IN:=FALSE;
	99:
		GapMove:=FALSE;
		GapState:=99;
		GapBusy:=FALSE;
		GapDone:=FALSE;
		Error:=TRUE;
		Top_MC_MoveAbsolute.Execute:=FALSE;
		Bottom_MC_MoveAbsolute.Execute:=FALSE;
		fb_ton.IN:=FALSE;
	-100:
		FB_PlcEmergencyStop();
		GapMove:=FALSE;
		GapState:=-100;
		GapBusy:=FALSE;
		GapDone:=FALSE;
		Error:=TRUE;
		Top_MC_MoveAbsolute.Execute:=FALSE;
		Bottom_MC_MoveAbsolute.Execute:=FALSE;
		fb_ton.IN:=FALSE;
END_CASE
END_IF
END_ACTION

ACTION A_LeftBottomMove:
IF LeftBottomMove THEN
LeftBottomBusy:=TRUE;
LeftBottomDone:=FALSE;
fb_ton_debug_3(PT:=t#10s);
(*×îºóÔÙ¼ì²éÒ»±éñîºÏ£¬²»ñîºÏÎªÕýÈ·×´Ì¬*)
IF LeftTopLin.NcToPlc.CoupleState<>0 OR LeftBottomLin.NcToPlc.CoupleState<>0
			OR RightTopLin.NcToPlc.CoupleState<>0 OR RightBottomLin.NcToPlc.CoupleState<>0 THEN
			ErrorID:=1;
			LeftBottomState:=-100;
END_IF
A_MoveMC();
CASE LeftBottomState OF
	0:
		IF Top_MC_MoveAbsolute.Error OR Bottom_MC_MoveAbsolute.Error
			OR RightTopLin_MC_MoveAbsolute.Error OR RightBottomLin_MC_MoveAbsolute.Error THEN		(*¼ì²éMC Error*)
			ErrorID:=2;
			LeftBottomState:=99;
		ELSIF leftTopLin.Status.NotMoving AND  leftBottomLin.Status.NotMoving
			 AND RightTopLin.Status.NotMoving AND RightBottomLin.Status.NotMoving THEN	(*Öá¶¼´¦ÓÚÍ£Ö¹×´Ì¬Ê±£¬×ªÏÂÒ»²½*)
			LeftBottomState:=1;
		END_IF
	1:
		Bottom_MC_MoveAbsolute.Position:=LeftBottomPosition;
		Bottom_MC_MoveAbsolute.Velocity:=LeftBottomVelocity;
		Bottom_MC_MoveAbsolute.Execute:=TRUE;
		fb_ton_debug_3.IN:=TRUE;
		LeftBottomState:=2;
	2:
		IF LeftTopLin.Status.Moving OR RightTopLin.Status.Moving OR RightBottomLin.Status.Moving THEN	(*³ýÁËÔË¶¯Öá¶¯£¬ÆäÓàÖáÓÐ¶¯£¬´íÎó*)
			ErrorID:=3;
			LeftBottomState:=-100;
		ELSIF NOT Bottom_MC_MoveAbsolute.Done THEN		(*ÔË¶¯ÖÐ£¬¼ì²éDoneÐÅºÅ£¬Ã»ÓÐÔòÑ­»·£¬³¬Ê±±¨´í*)
			(*IF NOT  fb_ton.Q THEN
				LeftBottomState:=2;
			ELSE
				ErrorID:=5;
				LeftBottomState:=-100;
			END_IF*)
			LeftBottomState:=2;
		ELSIF Bottom_MC_MoveAbsolute.Done THEN		(*ÔË¶¯Íê³É£¬×ªÏÂÒ»²½*)
				LeftBottomState:=88;
		END_IF
		(*½ÓÊÕµ½stopÐÅºÅÊ±£¬reset×´Ì¬*)
		IF LeftBottomReset THEN
			LeftBottomState:=89;
		END_IF

	88:
		LeftBottomMove:=FALSE;
		LeftBottomState:=0;
		LeftBottomBusy:=FALSE;
		LeftBottomDone:=TRUE;
		Error:=FALSE;
		ErrorID:=0;
		Bottom_MC_MoveAbsolute.Execute:=FALSE;
		fb_ton_debug_3.IN:=FALSE;
	89:
		LeftBottomMove:=FALSE;
		LeftBottomState:=0;
		LeftBottomBusy:=FALSE;
		LeftBottomDone:=FALSE;
		Error:=FALSE;
		ErrorID:=0;
		Bottom_MC_MoveAbsolute.Execute:=FALSE;
		fb_ton_debug_3.IN:=FALSE;
	99:
		LeftBottomMove:=FALSE;
		LeftBottomState:=99;
		LeftBottomBusy:=FALSE;
		LeftBottomDone:=FALSE;
		Error:=TRUE;
		Bottom_MC_MoveAbsolute.Execute:=FALSE;
		fb_ton_debug_3.IN:=FALSE;
	-100:
		FB_PlcEmergencyStop();
		LeftBottomMove:=FALSE;
		LeftBottomState:=-100;
		LeftBottomBusy:=FALSE;
		LeftBottomDone:=FALSE;
		Error:=TRUE;
		Bottom_MC_MoveAbsolute.Execute:=FALSE;
		fb_ton_debug_3.IN:=FALSE;
END_CASE
END_IF
END_ACTION

